DATA_BLOCK "G006G"
TITLE =
AUTHOR : KR
FAMILY : USW
VERSION : 0.0

"G006G_Code"
BEGIN
   Gr.FcCode := 0;
   Gr.Spare2 := 0;
   Gr.Spare4 := 0;
   Gr.Spare6 := 0;
   Gr.OutEmptyingTime := 0;
   Gr.ChangeBit.spare := B#16#0;
   Gr.ChangeBit.CBit1 := FALSE;
   Gr.ChangeBit.CBit2 := FALSE;
   Gr.ChangeBit.CBit3 := FALSE;
   Gr.ChangeBit.CBit4 := FALSE;
   Gr.StCode := 0;
   Gr.InEnableGr := FALSE;
   Gr.CmdContinue := FALSE;
   Gr.CmdRestartIdling := FALSE;
   Gr.InReleaseEmptyingTime := FALSE;
   Gr.InFeeding := FALSE;
   Gr.InOutAutostartMan := FALSE;
   Gr.InPreStart := FALSE;
   Gr.CmdManualOff := FALSE;
   Gr.CmdOff := FALSE;
   Gr.CmdOn := FALSE;
   Gr.CmdNext := FALSE;
   Gr.CmdFaultReset := FALSE;
   Gr.InOccupied := FALSE;
   Gr.InManual := FALSE;
   Gr.InLoadedSec := FALSE;
   Gr.InSeqStop := FALSE;
   Gr.ModePassive := FALSE;
   Gr.ModeActive := FALSE;
   Gr.ModeIdling := FALSE;
   Gr.spare163 := FALSE;
   Gr.spare164 := FALSE;
   Gr.spare165 := FALSE;
   Gr.spare166 := FALSE;
   Gr.spare167 := FALSE;
   Gr.StStopped := FALSE;
   Gr.StStarting := FALSE;
   Gr.StStarted := FALSE;
   Gr.StStopping := FALSE;
   Gr.StFault := FALSE;
   Gr.OutLoaded := FALSE;
   Gr.OutWarning := FALSE;
   Gr.OutFeeding := FALSE;
   Gr.OutEnableEl := FALSE;
   Gr.OutEnable1 := FALSE;
   Gr.OutHWStop := FALSE;
   Gr.OutDPFault := FALSE;
   Gr.OutAutostart := FALSE;
   Gr.OutManual := FALSE;
   Gr.OutHornOn := FALSE;
   Gr.OutEnablePrevGr := FALSE;
   Gr.VarStopped := FALSE;
   Gr.VarStarted := FALSE;
   Gr.VarFault := FALSE;
   Gr.VarStartwarning := FALSE;
   Gr.VarFlag1s := FALSE;
   Gr.OutEmptyingTimeDone := FALSE;
   Gr.OutNewWay := FALSE;
   Gr.OutSeqStop := FALSE;
   Gr.OutIdlingTime := 0;
   Gr.InCodePreselect := 0;
   Gr.InLine := 0;
   Gr.InCode := 0;
   Gr.OutCode := 0;
   Gr.Par.ParObjectNo := 0;
   Gr.Par.ParMgr := FALSE;
   Gr.Par.ParWgr := FALSE;
   Gr.Par.ParGgr := FALSE;
   Gr.Par.ParHornCode := 0;
   Gr.Par.ParIdling := 0;
   Gr.Par.ParEmptyingTime := 0;
   Gr.Par.Para1_0 := FALSE;
   Gr.Par.Para1_1 := FALSE;
   Gr.Par.Para1_2 := FALSE;
   Gr.Par.Para1_3 := FALSE;
   Gr.Par.Para1_4 := FALSE;
   Gr.Par.Para1_5 := FALSE;
   Gr.Par.Para1_6 := FALSE;
   Gr.Par.Para1_7 := FALSE;
   Gr.Par.Para1_8 := FALSE;
   Gr.Par.Para1_9 := FALSE;
   Gr.Par.Para1_10 := FALSE;
   Gr.Par.Para1_11 := FALSE;
   Gr.Par.Para1_12 := FALSE;
   Gr.Par.Para1_13 := FALSE;
   Gr.Par.Para1_14 := FALSE;
   Gr.Par.Para1_15 := FALSE;
   Gr.Par.Para2 := 0;
   Gr.Par.Para3 := 0;
   Gr.Par.Para4 := 0;
   Gr.Par.Para5 := 0;
   InOutValue1 := L#0;
   InOutValue2 := L#0;
   OutWayConflict := FALSE;
   OutSelectionOk := FALSE;
   CmdNewValue := FALSE;
   CmdNewJob := FALSE;
   OutCodeOK := FALSE;
   InEndOfJob := FALSE;
   staWayOk := FALSE;
   EdgeStartRelease := FALSE;
   USW8 := FALSE;
   USW9 := FALSE;
   USW10 := FALSE;
   USW11 := FALSE;
   USW12 := FALSE;
   USW13 := FALSE;
   USW14 := FALSE;
   USW15 := FALSE;
   A_1999_SHE01.StCode := 0;
   A_1999_SHE01.InMonTrue := FALSE;
   A_1999_SHE01.InMonFalse := FALSE;
   A_1999_SHE01.InPreAlarmTrue := FALSE;
   A_1999_SHE01.InPreAlarmFalse := FALSE;
   A_1999_SHE01.InStopTrueTime := FALSE;
   A_1999_SHE01.InStopFalseTime := FALSE;
   A_1999_SHE01.InpTrue := FALSE;
   A_1999_SHE01.InpFaultDev := FALSE;
   A_1999_SHE01.CmdRstTrueTime := FALSE;
   A_1999_SHE01.CmdRstFalseTime := FALSE;
   A_1999_SHE01.CmdRunTimeoutTime := FALSE;
   A_1999_SHE01.CmdFaultReset := FALSE;
   A_1999_SHE01.InLocal := FALSE;
   A_1999_SHE01.spare0305 := FALSE;
   A_1999_SHE01.InReport := FALSE;
   A_1999_SHE01.OutTimeoutTime := FALSE;
   A_1999_SHE01.InHWStop := FALSE;
   A_1999_SHE01.InDPFault := FALSE;
   A_1999_SHE01.OutPreAlarmTrue := FALSE;
   A_1999_SHE01.OutPreAlarmFalse := FALSE;
   A_1999_SHE01.OutFlagPos := FALSE;
   A_1999_SHE01.OutFlagNeg := FALSE;
   A_1999_SHE01.OutpFaultReset := FALSE;
   A_1999_SHE01.OutTrue := FALSE;
   A_1999_SHE01.StFalse := FALSE;
   A_1999_SHE01.StCtoTrue := FALSE;
   A_1999_SHE01.StTrue := FALSE;
   A_1999_SHE01.StCtoFalse := FALSE;
   A_1999_SHE01.StFault := FALSE;
   A_1999_SHE01.OutAlarmNrLog := 0;
   A_1999_SHE01.Par.ParObjectNo := 0;
   A_1999_SHE01.Par.ParMsgType := 0;
   A_1999_SHE01.Par.ParHornCode := 0;
   A_1999_SHE01.Par.ParLogOff := FALSE;
   A_1999_SHE01.Par.spare0401 := FALSE;
   A_1999_SHE01.Par.Par2WorkingCond := FALSE;
   A_1999_SHE01.Par.ParFaultRetry := FALSE;
   A_1999_SHE01.Par.ParBinLevel := FALSE;
   A_1999_SHE01.Par.ParDelayChange := 0;
   A_1999_SHE01.Par.ParDelayTrue := 0;
   A_1999_SHE01.Par.ParDelayFalse := 0;
   A_1999_SHE01.Par.ParTimeoutTrue := 0;
   A_1999_SHE01.Par.ParTimeoutFalse := 0;
   A_1999_SHE01.Par.OutMonTime := 0;
   A_1999_SHE01.Par.OutTransitionTime := 0;
   A_1999_SHE01.Par.OutMonTrue := FALSE;
   A_1999_SHE01.Par.OutMonFalse := FALSE;
   A_1999_SHE01.Par.OutFlagFaultDev := FALSE;
   A_1999_SHE01.Par.OutDelayTime := 0;
   A_1999_SHE02.StCode := 0;
   A_1999_SHE02.InMonTrue := FALSE;
   A_1999_SHE02.InMonFalse := FALSE;
   A_1999_SHE02.InPreAlarmTrue := FALSE;
   A_1999_SHE02.InPreAlarmFalse := FALSE;
   A_1999_SHE02.InStopTrueTime := FALSE;
   A_1999_SHE02.InStopFalseTime := FALSE;
   A_1999_SHE02.InpTrue := FALSE;
   A_1999_SHE02.InpFaultDev := FALSE;
   A_1999_SHE02.CmdRstTrueTime := FALSE;
   A_1999_SHE02.CmdRstFalseTime := FALSE;
   A_1999_SHE02.CmdRunTimeoutTime := FALSE;
   A_1999_SHE02.CmdFaultReset := FALSE;
   A_1999_SHE02.InLocal := FALSE;
   A_1999_SHE02.spare0305 := FALSE;
   A_1999_SHE02.InReport := FALSE;
   A_1999_SHE02.OutTimeoutTime := FALSE;
   A_1999_SHE02.InHWStop := FALSE;
   A_1999_SHE02.InDPFault := FALSE;
   A_1999_SHE02.OutPreAlarmTrue := FALSE;
   A_1999_SHE02.OutPreAlarmFalse := FALSE;
   A_1999_SHE02.OutFlagPos := FALSE;
   A_1999_SHE02.OutFlagNeg := FALSE;
   A_1999_SHE02.OutpFaultReset := FALSE;
   A_1999_SHE02.OutTrue := FALSE;
   A_1999_SHE02.StFalse := FALSE;
   A_1999_SHE02.StCtoTrue := FALSE;
   A_1999_SHE02.StTrue := FALSE;
   A_1999_SHE02.StCtoFalse := FALSE;
   A_1999_SHE02.StFault := FALSE;
   A_1999_SHE02.OutAlarmNrLog := 0;
   A_1999_SHE02.Par.ParObjectNo := 0;
   A_1999_SHE02.Par.ParMsgType := 0;
   A_1999_SHE02.Par.ParHornCode := 0;
   A_1999_SHE02.Par.ParLogOff := FALSE;
   A_1999_SHE02.Par.spare0401 := FALSE;
   A_1999_SHE02.Par.Par2WorkingCond := FALSE;
   A_1999_SHE02.Par.ParFaultRetry := FALSE;
   A_1999_SHE02.Par.ParBinLevel := FALSE;
   A_1999_SHE02.Par.ParDelayChange := 0;
   A_1999_SHE02.Par.ParDelayTrue := 0;
   A_1999_SHE02.Par.ParDelayFalse := 0;
   A_1999_SHE02.Par.ParTimeoutTrue := 0;
   A_1999_SHE02.Par.ParTimeoutFalse := 0;
   A_1999_SHE02.Par.OutMonTime := 0;
   A_1999_SHE02.Par.OutTransitionTime := 0;
   A_1999_SHE02.Par.OutMonTrue := FALSE;
   A_1999_SHE02.Par.OutMonFalse := FALSE;
   A_1999_SHE02.Par.OutFlagFaultDev := FALSE;
   A_1999_SHE02.Par.OutDelayTime := 0;
   A_19_A040Z1.StCode := 0;
   A_19_A040Z1.InMonTrue := FALSE;
   A_19_A040Z1.InMonFalse := FALSE;
   A_19_A040Z1.InPreAlarmTrue := FALSE;
   A_19_A040Z1.InPreAlarmFalse := FALSE;
   A_19_A040Z1.InStopTrueTime := FALSE;
   A_19_A040Z1.InStopFalseTime := FALSE;
   A_19_A040Z1.InpTrue := FALSE;
   A_19_A040Z1.InpFaultDev := FALSE;
   A_19_A040Z1.CmdRstTrueTime := FALSE;
   A_19_A040Z1.CmdRstFalseTime := FALSE;
   A_19_A040Z1.CmdRunTimeoutTime := FALSE;
   A_19_A040Z1.CmdFaultReset := FALSE;
   A_19_A040Z1.InLocal := FALSE;
   A_19_A040Z1.spare0305 := FALSE;
   A_19_A040Z1.InReport := FALSE;
   A_19_A040Z1.OutTimeoutTime := FALSE;
   A_19_A040Z1.InHWStop := FALSE;
   A_19_A040Z1.InDPFault := FALSE;
   A_19_A040Z1.OutPreAlarmTrue := FALSE;
   A_19_A040Z1.OutPreAlarmFalse := FALSE;
   A_19_A040Z1.OutFlagPos := FALSE;
   A_19_A040Z1.OutFlagNeg := FALSE;
   A_19_A040Z1.OutpFaultReset := FALSE;
   A_19_A040Z1.OutTrue := FALSE;
   A_19_A040Z1.StFalse := FALSE;
   A_19_A040Z1.StCtoTrue := FALSE;
   A_19_A040Z1.StTrue := FALSE;
   A_19_A040Z1.StCtoFalse := FALSE;
   A_19_A040Z1.StFault := FALSE;
   A_19_A040Z1.OutAlarmNrLog := 0;
   A_19_A040Z1.Par.ParObjectNo := 0;
   A_19_A040Z1.Par.ParMsgType := 0;
   A_19_A040Z1.Par.ParHornCode := 0;
   A_19_A040Z1.Par.ParLogOff := FALSE;
   A_19_A040Z1.Par.spare0401 := FALSE;
   A_19_A040Z1.Par.Par2WorkingCond := FALSE;
   A_19_A040Z1.Par.ParFaultRetry := FALSE;
   A_19_A040Z1.Par.ParBinLevel := FALSE;
   A_19_A040Z1.Par.ParDelayChange := 0;
   A_19_A040Z1.Par.ParDelayTrue := 0;
   A_19_A040Z1.Par.ParDelayFalse := 0;
   A_19_A040Z1.Par.ParTimeoutTrue := 0;
   A_19_A040Z1.Par.ParTimeoutFalse := 0;
   A_19_A040Z1.Par.OutMonTime := 0;
   A_19_A040Z1.Par.OutTransitionTime := 0;
   A_19_A040Z1.Par.OutMonTrue := FALSE;
   A_19_A040Z1.Par.OutMonFalse := FALSE;
   A_19_A040Z1.Par.OutFlagFaultDev := FALSE;
   A_19_A040Z1.Par.OutDelayTime := 0;
   A_19_A097Z1.StCode := 0;
   A_19_A097Z1.InMonTrue := FALSE;
   A_19_A097Z1.InMonFalse := FALSE;
   A_19_A097Z1.InPreAlarmTrue := FALSE;
   A_19_A097Z1.InPreAlarmFalse := FALSE;
   A_19_A097Z1.InStopTrueTime := FALSE;
   A_19_A097Z1.InStopFalseTime := FALSE;
   A_19_A097Z1.InpTrue := FALSE;
   A_19_A097Z1.InpFaultDev := FALSE;
   A_19_A097Z1.CmdRstTrueTime := FALSE;
   A_19_A097Z1.CmdRstFalseTime := FALSE;
   A_19_A097Z1.CmdRunTimeoutTime := FALSE;
   A_19_A097Z1.CmdFaultReset := FALSE;
   A_19_A097Z1.InLocal := FALSE;
   A_19_A097Z1.spare0305 := FALSE;
   A_19_A097Z1.InReport := FALSE;
   A_19_A097Z1.OutTimeoutTime := FALSE;
   A_19_A097Z1.InHWStop := FALSE;
   A_19_A097Z1.InDPFault := FALSE;
   A_19_A097Z1.OutPreAlarmTrue := FALSE;
   A_19_A097Z1.OutPreAlarmFalse := FALSE;
   A_19_A097Z1.OutFlagPos := FALSE;
   A_19_A097Z1.OutFlagNeg := FALSE;
   A_19_A097Z1.OutpFaultReset := FALSE;
   A_19_A097Z1.OutTrue := FALSE;
   A_19_A097Z1.StFalse := FALSE;
   A_19_A097Z1.StCtoTrue := FALSE;
   A_19_A097Z1.StTrue := FALSE;
   A_19_A097Z1.StCtoFalse := FALSE;
   A_19_A097Z1.StFault := FALSE;
   A_19_A097Z1.OutAlarmNrLog := 0;
   A_19_A097Z1.Par.ParObjectNo := 0;
   A_19_A097Z1.Par.ParMsgType := 0;
   A_19_A097Z1.Par.ParHornCode := 0;
   A_19_A097Z1.Par.ParLogOff := FALSE;
   A_19_A097Z1.Par.spare0401 := FALSE;
   A_19_A097Z1.Par.Par2WorkingCond := FALSE;
   A_19_A097Z1.Par.ParFaultRetry := FALSE;
   A_19_A097Z1.Par.ParBinLevel := FALSE;
   A_19_A097Z1.Par.ParDelayChange := 0;
   A_19_A097Z1.Par.ParDelayTrue := 0;
   A_19_A097Z1.Par.ParDelayFalse := 0;
   A_19_A097Z1.Par.ParTimeoutTrue := 0;
   A_19_A097Z1.Par.ParTimeoutFalse := 0;
   A_19_A097Z1.Par.OutMonTime := 0;
   A_19_A097Z1.Par.OutTransitionTime := 0;
   A_19_A097Z1.Par.OutMonTrue := FALSE;
   A_19_A097Z1.Par.OutMonFalse := FALSE;
   A_19_A097Z1.Par.OutFlagFaultDev := FALSE;
   A_19_A097Z1.Par.OutDelayTime := 0;
   A_19_K091Z1.StCode := 0;
   A_19_K091Z1.InMonTrue := FALSE;
   A_19_K091Z1.InMonFalse := FALSE;
   A_19_K091Z1.InPreAlarmTrue := FALSE;
   A_19_K091Z1.InPreAlarmFalse := FALSE;
   A_19_K091Z1.InStopTrueTime := FALSE;
   A_19_K091Z1.InStopFalseTime := FALSE;
   A_19_K091Z1.InpTrue := FALSE;
   A_19_K091Z1.InpFaultDev := FALSE;
   A_19_K091Z1.CmdRstTrueTime := FALSE;
   A_19_K091Z1.CmdRstFalseTime := FALSE;
   A_19_K091Z1.CmdRunTimeoutTime := FALSE;
   A_19_K091Z1.CmdFaultReset := FALSE;
   A_19_K091Z1.InLocal := FALSE;
   A_19_K091Z1.spare0305 := FALSE;
   A_19_K091Z1.InReport := FALSE;
   A_19_K091Z1.OutTimeoutTime := FALSE;
   A_19_K091Z1.InHWStop := FALSE;
   A_19_K091Z1.InDPFault := FALSE;
   A_19_K091Z1.OutPreAlarmTrue := FALSE;
   A_19_K091Z1.OutPreAlarmFalse := FALSE;
   A_19_K091Z1.OutFlagPos := FALSE;
   A_19_K091Z1.OutFlagNeg := FALSE;
   A_19_K091Z1.OutpFaultReset := FALSE;
   A_19_K091Z1.OutTrue := FALSE;
   A_19_K091Z1.StFalse := FALSE;
   A_19_K091Z1.StCtoTrue := FALSE;
   A_19_K091Z1.StTrue := FALSE;
   A_19_K091Z1.StCtoFalse := FALSE;
   A_19_K091Z1.StFault := FALSE;
   A_19_K091Z1.OutAlarmNrLog := 0;
   A_19_K091Z1.Par.ParObjectNo := 0;
   A_19_K091Z1.Par.ParMsgType := 0;
   A_19_K091Z1.Par.ParHornCode := 0;
   A_19_K091Z1.Par.ParLogOff := FALSE;
   A_19_K091Z1.Par.spare0401 := FALSE;
   A_19_K091Z1.Par.Par2WorkingCond := FALSE;
   A_19_K091Z1.Par.ParFaultRetry := FALSE;
   A_19_K091Z1.Par.ParBinLevel := FALSE;
   A_19_K091Z1.Par.ParDelayChange := 0;
   A_19_K091Z1.Par.ParDelayTrue := 0;
   A_19_K091Z1.Par.ParDelayFalse := 0;
   A_19_K091Z1.Par.ParTimeoutTrue := 0;
   A_19_K091Z1.Par.ParTimeoutFalse := 0;
   A_19_K091Z1.Par.OutMonTime := 0;
   A_19_K091Z1.Par.OutTransitionTime := 0;
   A_19_K091Z1.Par.OutMonTrue := FALSE;
   A_19_K091Z1.Par.OutMonFalse := FALSE;
   A_19_K091Z1.Par.OutFlagFaultDev := FALSE;
   A_19_K091Z1.Par.OutDelayTime := 0;
   A_19_S_H097Z1.StCode := 0;
   A_19_S_H097Z1.InMonTrue := FALSE;
   A_19_S_H097Z1.InMonFalse := FALSE;
   A_19_S_H097Z1.InPreAlarmTrue := FALSE;
   A_19_S_H097Z1.InPreAlarmFalse := FALSE;
   A_19_S_H097Z1.InStopTrueTime := FALSE;
   A_19_S_H097Z1.InStopFalseTime := FALSE;
   A_19_S_H097Z1.InpTrue := FALSE;
   A_19_S_H097Z1.InpFaultDev := FALSE;
   A_19_S_H097Z1.CmdRstTrueTime := FALSE;
   A_19_S_H097Z1.CmdRstFalseTime := FALSE;
   A_19_S_H097Z1.CmdRunTimeoutTime := FALSE;
   A_19_S_H097Z1.CmdFaultReset := FALSE;
   A_19_S_H097Z1.InLocal := FALSE;
   A_19_S_H097Z1.spare0305 := FALSE;
   A_19_S_H097Z1.InReport := FALSE;
   A_19_S_H097Z1.OutTimeoutTime := FALSE;
   A_19_S_H097Z1.InHWStop := FALSE;
   A_19_S_H097Z1.InDPFault := FALSE;
   A_19_S_H097Z1.OutPreAlarmTrue := FALSE;
   A_19_S_H097Z1.OutPreAlarmFalse := FALSE;
   A_19_S_H097Z1.OutFlagPos := FALSE;
   A_19_S_H097Z1.OutFlagNeg := FALSE;
   A_19_S_H097Z1.OutpFaultReset := FALSE;
   A_19_S_H097Z1.OutTrue := FALSE;
   A_19_S_H097Z1.StFalse := FALSE;
   A_19_S_H097Z1.StCtoTrue := FALSE;
   A_19_S_H097Z1.StTrue := FALSE;
   A_19_S_H097Z1.StCtoFalse := FALSE;
   A_19_S_H097Z1.StFault := FALSE;
   A_19_S_H097Z1.OutAlarmNrLog := 0;
   A_19_S_H097Z1.Par.ParObjectNo := 0;
   A_19_S_H097Z1.Par.ParMsgType := 0;
   A_19_S_H097Z1.Par.ParHornCode := 0;
   A_19_S_H097Z1.Par.ParLogOff := FALSE;
   A_19_S_H097Z1.Par.spare0401 := FALSE;
   A_19_S_H097Z1.Par.Par2WorkingCond := FALSE;
   A_19_S_H097Z1.Par.ParFaultRetry := FALSE;
   A_19_S_H097Z1.Par.ParBinLevel := FALSE;
   A_19_S_H097Z1.Par.ParDelayChange := 0;
   A_19_S_H097Z1.Par.ParDelayTrue := 0;
   A_19_S_H097Z1.Par.ParDelayFalse := 0;
   A_19_S_H097Z1.Par.ParTimeoutTrue := 0;
   A_19_S_H097Z1.Par.ParTimeoutFalse := 0;
   A_19_S_H097Z1.Par.OutMonTime := 0;
   A_19_S_H097Z1.Par.OutTransitionTime := 0;
   A_19_S_H097Z1.Par.OutMonTrue := FALSE;
   A_19_S_H097Z1.Par.OutMonFalse := FALSE;
   A_19_S_H097Z1.Par.OutFlagFaultDev := FALSE;
   A_19_S_H097Z1.Par.OutDelayTime := 0;
   A_2201_SHE20.StCode := 0;
   A_2201_SHE20.InMonTrue := FALSE;
   A_2201_SHE20.InMonFalse := FALSE;
   A_2201_SHE20.InPreAlarmTrue := FALSE;
   A_2201_SHE20.InPreAlarmFalse := FALSE;
   A_2201_SHE20.InStopTrueTime := FALSE;
   A_2201_SHE20.InStopFalseTime := FALSE;
   A_2201_SHE20.InpTrue := FALSE;
   A_2201_SHE20.InpFaultDev := FALSE;
   A_2201_SHE20.CmdRstTrueTime := FALSE;
   A_2201_SHE20.CmdRstFalseTime := FALSE;
   A_2201_SHE20.CmdRunTimeoutTime := FALSE;
   A_2201_SHE20.CmdFaultReset := FALSE;
   A_2201_SHE20.InLocal := FALSE;
   A_2201_SHE20.spare0305 := FALSE;
   A_2201_SHE20.InReport := FALSE;
   A_2201_SHE20.OutTimeoutTime := FALSE;
   A_2201_SHE20.InHWStop := FALSE;
   A_2201_SHE20.InDPFault := FALSE;
   A_2201_SHE20.OutPreAlarmTrue := FALSE;
   A_2201_SHE20.OutPreAlarmFalse := FALSE;
   A_2201_SHE20.OutFlagPos := FALSE;
   A_2201_SHE20.OutFlagNeg := FALSE;
   A_2201_SHE20.OutpFaultReset := FALSE;
   A_2201_SHE20.OutTrue := FALSE;
   A_2201_SHE20.StFalse := FALSE;
   A_2201_SHE20.StCtoTrue := FALSE;
   A_2201_SHE20.StTrue := FALSE;
   A_2201_SHE20.StCtoFalse := FALSE;
   A_2201_SHE20.StFault := FALSE;
   A_2201_SHE20.OutAlarmNrLog := 0;
   A_2201_SHE20.Par.ParObjectNo := 0;
   A_2201_SHE20.Par.ParMsgType := 0;
   A_2201_SHE20.Par.ParHornCode := 0;
   A_2201_SHE20.Par.ParLogOff := FALSE;
   A_2201_SHE20.Par.spare0401 := FALSE;
   A_2201_SHE20.Par.Par2WorkingCond := FALSE;
   A_2201_SHE20.Par.ParFaultRetry := FALSE;
   A_2201_SHE20.Par.ParBinLevel := FALSE;
   A_2201_SHE20.Par.ParDelayChange := 0;
   A_2201_SHE20.Par.ParDelayTrue := 0;
   A_2201_SHE20.Par.ParDelayFalse := 0;
   A_2201_SHE20.Par.ParTimeoutTrue := 0;
   A_2201_SHE20.Par.ParTimeoutFalse := 0;
   A_2201_SHE20.Par.OutMonTime := 0;
   A_2201_SHE20.Par.OutTransitionTime := 0;
   A_2201_SHE20.Par.OutMonTrue := FALSE;
   A_2201_SHE20.Par.OutMonFalse := FALSE;
   A_2201_SHE20.Par.OutFlagFaultDev := FALSE;
   A_2201_SHE20.Par.OutDelayTime := 0;
   A_2201_SHE21.StCode := 0;
   A_2201_SHE21.InMonTrue := FALSE;
   A_2201_SHE21.InMonFalse := FALSE;
   A_2201_SHE21.InPreAlarmTrue := FALSE;
   A_2201_SHE21.InPreAlarmFalse := FALSE;
   A_2201_SHE21.InStopTrueTime := FALSE;
   A_2201_SHE21.InStopFalseTime := FALSE;
   A_2201_SHE21.InpTrue := FALSE;
   A_2201_SHE21.InpFaultDev := FALSE;
   A_2201_SHE21.CmdRstTrueTime := FALSE;
   A_2201_SHE21.CmdRstFalseTime := FALSE;
   A_2201_SHE21.CmdRunTimeoutTime := FALSE;
   A_2201_SHE21.CmdFaultReset := FALSE;
   A_2201_SHE21.InLocal := FALSE;
   A_2201_SHE21.spare0305 := FALSE;
   A_2201_SHE21.InReport := FALSE;
   A_2201_SHE21.OutTimeoutTime := FALSE;
   A_2201_SHE21.InHWStop := FALSE;
   A_2201_SHE21.InDPFault := FALSE;
   A_2201_SHE21.OutPreAlarmTrue := FALSE;
   A_2201_SHE21.OutPreAlarmFalse := FALSE;
   A_2201_SHE21.OutFlagPos := FALSE;
   A_2201_SHE21.OutFlagNeg := FALSE;
   A_2201_SHE21.OutpFaultReset := FALSE;
   A_2201_SHE21.OutTrue := FALSE;
   A_2201_SHE21.StFalse := FALSE;
   A_2201_SHE21.StCtoTrue := FALSE;
   A_2201_SHE21.StTrue := FALSE;
   A_2201_SHE21.StCtoFalse := FALSE;
   A_2201_SHE21.StFault := FALSE;
   A_2201_SHE21.OutAlarmNrLog := 0;
   A_2201_SHE21.Par.ParObjectNo := 0;
   A_2201_SHE21.Par.ParMsgType := 0;
   A_2201_SHE21.Par.ParHornCode := 0;
   A_2201_SHE21.Par.ParLogOff := FALSE;
   A_2201_SHE21.Par.spare0401 := FALSE;
   A_2201_SHE21.Par.Par2WorkingCond := FALSE;
   A_2201_SHE21.Par.ParFaultRetry := FALSE;
   A_2201_SHE21.Par.ParBinLevel := FALSE;
   A_2201_SHE21.Par.ParDelayChange := 0;
   A_2201_SHE21.Par.ParDelayTrue := 0;
   A_2201_SHE21.Par.ParDelayFalse := 0;
   A_2201_SHE21.Par.ParTimeoutTrue := 0;
   A_2201_SHE21.Par.ParTimeoutFalse := 0;
   A_2201_SHE21.Par.OutMonTime := 0;
   A_2201_SHE21.Par.OutTransitionTime := 0;
   A_2201_SHE21.Par.OutMonTrue := FALSE;
   A_2201_SHE21.Par.OutMonFalse := FALSE;
   A_2201_SHE21.Par.OutFlagFaultDev := FALSE;
   A_2201_SHE21.Par.OutDelayTime := 0;
   A_2201_SHE22.StCode := 0;
   A_2201_SHE22.InMonTrue := FALSE;
   A_2201_SHE22.InMonFalse := FALSE;
   A_2201_SHE22.InPreAlarmTrue := FALSE;
   A_2201_SHE22.InPreAlarmFalse := FALSE;
   A_2201_SHE22.InStopTrueTime := FALSE;
   A_2201_SHE22.InStopFalseTime := FALSE;
   A_2201_SHE22.InpTrue := FALSE;
   A_2201_SHE22.InpFaultDev := FALSE;
   A_2201_SHE22.CmdRstTrueTime := FALSE;
   A_2201_SHE22.CmdRstFalseTime := FALSE;
   A_2201_SHE22.CmdRunTimeoutTime := FALSE;
   A_2201_SHE22.CmdFaultReset := FALSE;
   A_2201_SHE22.InLocal := FALSE;
   A_2201_SHE22.spare0305 := FALSE;
   A_2201_SHE22.InReport := FALSE;
   A_2201_SHE22.OutTimeoutTime := FALSE;
   A_2201_SHE22.InHWStop := FALSE;
   A_2201_SHE22.InDPFault := FALSE;
   A_2201_SHE22.OutPreAlarmTrue := FALSE;
   A_2201_SHE22.OutPreAlarmFalse := FALSE;
   A_2201_SHE22.OutFlagPos := FALSE;
   A_2201_SHE22.OutFlagNeg := FALSE;
   A_2201_SHE22.OutpFaultReset := FALSE;
   A_2201_SHE22.OutTrue := FALSE;
   A_2201_SHE22.StFalse := FALSE;
   A_2201_SHE22.StCtoTrue := FALSE;
   A_2201_SHE22.StTrue := FALSE;
   A_2201_SHE22.StCtoFalse := FALSE;
   A_2201_SHE22.StFault := FALSE;
   A_2201_SHE22.OutAlarmNrLog := 0;
   A_2201_SHE22.Par.ParObjectNo := 0;
   A_2201_SHE22.Par.ParMsgType := 0;
   A_2201_SHE22.Par.ParHornCode := 0;
   A_2201_SHE22.Par.ParLogOff := FALSE;
   A_2201_SHE22.Par.spare0401 := FALSE;
   A_2201_SHE22.Par.Par2WorkingCond := FALSE;
   A_2201_SHE22.Par.ParFaultRetry := FALSE;
   A_2201_SHE22.Par.ParBinLevel := FALSE;
   A_2201_SHE22.Par.ParDelayChange := 0;
   A_2201_SHE22.Par.ParDelayTrue := 0;
   A_2201_SHE22.Par.ParDelayFalse := 0;
   A_2201_SHE22.Par.ParTimeoutTrue := 0;
   A_2201_SHE22.Par.ParTimeoutFalse := 0;
   A_2201_SHE22.Par.OutMonTime := 0;
   A_2201_SHE22.Par.OutTransitionTime := 0;
   A_2201_SHE22.Par.OutMonTrue := FALSE;
   A_2201_SHE22.Par.OutMonFalse := FALSE;
   A_2201_SHE22.Par.OutFlagFaultDev := FALSE;
   A_2201_SHE22.Par.OutDelayTime := 0;
   A_2201_SHE23.StCode := 0;
   A_2201_SHE23.InMonTrue := FALSE;
   A_2201_SHE23.InMonFalse := FALSE;
   A_2201_SHE23.InPreAlarmTrue := FALSE;
   A_2201_SHE23.InPreAlarmFalse := FALSE;
   A_2201_SHE23.InStopTrueTime := FALSE;
   A_2201_SHE23.InStopFalseTime := FALSE;
   A_2201_SHE23.InpTrue := FALSE;
   A_2201_SHE23.InpFaultDev := FALSE;
   A_2201_SHE23.CmdRstTrueTime := FALSE;
   A_2201_SHE23.CmdRstFalseTime := FALSE;
   A_2201_SHE23.CmdRunTimeoutTime := FALSE;
   A_2201_SHE23.CmdFaultReset := FALSE;
   A_2201_SHE23.InLocal := FALSE;
   A_2201_SHE23.spare0305 := FALSE;
   A_2201_SHE23.InReport := FALSE;
   A_2201_SHE23.OutTimeoutTime := FALSE;
   A_2201_SHE23.InHWStop := FALSE;
   A_2201_SHE23.InDPFault := FALSE;
   A_2201_SHE23.OutPreAlarmTrue := FALSE;
   A_2201_SHE23.OutPreAlarmFalse := FALSE;
   A_2201_SHE23.OutFlagPos := FALSE;
   A_2201_SHE23.OutFlagNeg := FALSE;
   A_2201_SHE23.OutpFaultReset := FALSE;
   A_2201_SHE23.OutTrue := FALSE;
   A_2201_SHE23.StFalse := FALSE;
   A_2201_SHE23.StCtoTrue := FALSE;
   A_2201_SHE23.StTrue := FALSE;
   A_2201_SHE23.StCtoFalse := FALSE;
   A_2201_SHE23.StFault := FALSE;
   A_2201_SHE23.OutAlarmNrLog := 0;
   A_2201_SHE23.Par.ParObjectNo := 0;
   A_2201_SHE23.Par.ParMsgType := 0;
   A_2201_SHE23.Par.ParHornCode := 0;
   A_2201_SHE23.Par.ParLogOff := FALSE;
   A_2201_SHE23.Par.spare0401 := FALSE;
   A_2201_SHE23.Par.Par2WorkingCond := FALSE;
   A_2201_SHE23.Par.ParFaultRetry := FALSE;
   A_2201_SHE23.Par.ParBinLevel := FALSE;
   A_2201_SHE23.Par.ParDelayChange := 0;
   A_2201_SHE23.Par.ParDelayTrue := 0;
   A_2201_SHE23.Par.ParDelayFalse := 0;
   A_2201_SHE23.Par.ParTimeoutTrue := 0;
   A_2201_SHE23.Par.ParTimeoutFalse := 0;
   A_2201_SHE23.Par.OutMonTime := 0;
   A_2201_SHE23.Par.OutTransitionTime := 0;
   A_2201_SHE23.Par.OutMonTrue := FALSE;
   A_2201_SHE23.Par.OutMonFalse := FALSE;
   A_2201_SHE23.Par.OutFlagFaultDev := FALSE;
   A_2201_SHE23.Par.OutDelayTime := 0;
   A_2299_SHE01.StCode := 0;
   A_2299_SHE01.InMonTrue := FALSE;
   A_2299_SHE01.InMonFalse := FALSE;
   A_2299_SHE01.InPreAlarmTrue := FALSE;
   A_2299_SHE01.InPreAlarmFalse := FALSE;
   A_2299_SHE01.InStopTrueTime := FALSE;
   A_2299_SHE01.InStopFalseTime := FALSE;
   A_2299_SHE01.InpTrue := FALSE;
   A_2299_SHE01.InpFaultDev := FALSE;
   A_2299_SHE01.CmdRstTrueTime := FALSE;
   A_2299_SHE01.CmdRstFalseTime := FALSE;
   A_2299_SHE01.CmdRunTimeoutTime := FALSE;
   A_2299_SHE01.CmdFaultReset := FALSE;
   A_2299_SHE01.InLocal := FALSE;
   A_2299_SHE01.spare0305 := FALSE;
   A_2299_SHE01.InReport := FALSE;
   A_2299_SHE01.OutTimeoutTime := FALSE;
   A_2299_SHE01.InHWStop := FALSE;
   A_2299_SHE01.InDPFault := FALSE;
   A_2299_SHE01.OutPreAlarmTrue := FALSE;
   A_2299_SHE01.OutPreAlarmFalse := FALSE;
   A_2299_SHE01.OutFlagPos := FALSE;
   A_2299_SHE01.OutFlagNeg := FALSE;
   A_2299_SHE01.OutpFaultReset := FALSE;
   A_2299_SHE01.OutTrue := FALSE;
   A_2299_SHE01.StFalse := FALSE;
   A_2299_SHE01.StCtoTrue := FALSE;
   A_2299_SHE01.StTrue := FALSE;
   A_2299_SHE01.StCtoFalse := FALSE;
   A_2299_SHE01.StFault := FALSE;
   A_2299_SHE01.OutAlarmNrLog := 0;
   A_2299_SHE01.Par.ParObjectNo := 0;
   A_2299_SHE01.Par.ParMsgType := 0;
   A_2299_SHE01.Par.ParHornCode := 0;
   A_2299_SHE01.Par.ParLogOff := FALSE;
   A_2299_SHE01.Par.spare0401 := FALSE;
   A_2299_SHE01.Par.Par2WorkingCond := FALSE;
   A_2299_SHE01.Par.ParFaultRetry := FALSE;
   A_2299_SHE01.Par.ParBinLevel := FALSE;
   A_2299_SHE01.Par.ParDelayChange := 0;
   A_2299_SHE01.Par.ParDelayTrue := 0;
   A_2299_SHE01.Par.ParDelayFalse := 0;
   A_2299_SHE01.Par.ParTimeoutTrue := 0;
   A_2299_SHE01.Par.ParTimeoutFalse := 0;
   A_2299_SHE01.Par.OutMonTime := 0;
   A_2299_SHE01.Par.OutTransitionTime := 0;
   A_2299_SHE01.Par.OutMonTrue := FALSE;
   A_2299_SHE01.Par.OutMonFalse := FALSE;
   A_2299_SHE01.Par.OutFlagFaultDev := FALSE;
   A_2299_SHE01.Par.OutDelayTime := 0;
   A_2299_SHE02.StCode := 0;
   A_2299_SHE02.InMonTrue := FALSE;
   A_2299_SHE02.InMonFalse := FALSE;
   A_2299_SHE02.InPreAlarmTrue := FALSE;
   A_2299_SHE02.InPreAlarmFalse := FALSE;
   A_2299_SHE02.InStopTrueTime := FALSE;
   A_2299_SHE02.InStopFalseTime := FALSE;
   A_2299_SHE02.InpTrue := FALSE;
   A_2299_SHE02.InpFaultDev := FALSE;
   A_2299_SHE02.CmdRstTrueTime := FALSE;
   A_2299_SHE02.CmdRstFalseTime := FALSE;
   A_2299_SHE02.CmdRunTimeoutTime := FALSE;
   A_2299_SHE02.CmdFaultReset := FALSE;
   A_2299_SHE02.InLocal := FALSE;
   A_2299_SHE02.spare0305 := FALSE;
   A_2299_SHE02.InReport := FALSE;
   A_2299_SHE02.OutTimeoutTime := FALSE;
   A_2299_SHE02.InHWStop := FALSE;
   A_2299_SHE02.InDPFault := FALSE;
   A_2299_SHE02.OutPreAlarmTrue := FALSE;
   A_2299_SHE02.OutPreAlarmFalse := FALSE;
   A_2299_SHE02.OutFlagPos := FALSE;
   A_2299_SHE02.OutFlagNeg := FALSE;
   A_2299_SHE02.OutpFaultReset := FALSE;
   A_2299_SHE02.OutTrue := FALSE;
   A_2299_SHE02.StFalse := FALSE;
   A_2299_SHE02.StCtoTrue := FALSE;
   A_2299_SHE02.StTrue := FALSE;
   A_2299_SHE02.StCtoFalse := FALSE;
   A_2299_SHE02.StFault := FALSE;
   A_2299_SHE02.OutAlarmNrLog := 0;
   A_2299_SHE02.Par.ParObjectNo := 0;
   A_2299_SHE02.Par.ParMsgType := 0;
   A_2299_SHE02.Par.ParHornCode := 0;
   A_2299_SHE02.Par.ParLogOff := FALSE;
   A_2299_SHE02.Par.spare0401 := FALSE;
   A_2299_SHE02.Par.Par2WorkingCond := FALSE;
   A_2299_SHE02.Par.ParFaultRetry := FALSE;
   A_2299_SHE02.Par.ParBinLevel := FALSE;
   A_2299_SHE02.Par.ParDelayChange := 0;
   A_2299_SHE02.Par.ParDelayTrue := 0;
   A_2299_SHE02.Par.ParDelayFalse := 0;
   A_2299_SHE02.Par.ParTimeoutTrue := 0;
   A_2299_SHE02.Par.ParTimeoutFalse := 0;
   A_2299_SHE02.Par.OutMonTime := 0;
   A_2299_SHE02.Par.OutTransitionTime := 0;
   A_2299_SHE02.Par.OutMonTrue := FALSE;
   A_2299_SHE02.Par.OutMonFalse := FALSE;
   A_2299_SHE02.Par.OutFlagFaultDev := FALSE;
   A_2299_SHE02.Par.OutDelayTime := 0;
   A_2299_SHE03.StCode := 0;
   A_2299_SHE03.InMonTrue := FALSE;
   A_2299_SHE03.InMonFalse := FALSE;
   A_2299_SHE03.InPreAlarmTrue := FALSE;
   A_2299_SHE03.InPreAlarmFalse := FALSE;
   A_2299_SHE03.InStopTrueTime := FALSE;
   A_2299_SHE03.InStopFalseTime := FALSE;
   A_2299_SHE03.InpTrue := FALSE;
   A_2299_SHE03.InpFaultDev := FALSE;
   A_2299_SHE03.CmdRstTrueTime := FALSE;
   A_2299_SHE03.CmdRstFalseTime := FALSE;
   A_2299_SHE03.CmdRunTimeoutTime := FALSE;
   A_2299_SHE03.CmdFaultReset := FALSE;
   A_2299_SHE03.InLocal := FALSE;
   A_2299_SHE03.spare0305 := FALSE;
   A_2299_SHE03.InReport := FALSE;
   A_2299_SHE03.OutTimeoutTime := FALSE;
   A_2299_SHE03.InHWStop := FALSE;
   A_2299_SHE03.InDPFault := FALSE;
   A_2299_SHE03.OutPreAlarmTrue := FALSE;
   A_2299_SHE03.OutPreAlarmFalse := FALSE;
   A_2299_SHE03.OutFlagPos := FALSE;
   A_2299_SHE03.OutFlagNeg := FALSE;
   A_2299_SHE03.OutpFaultReset := FALSE;
   A_2299_SHE03.OutTrue := FALSE;
   A_2299_SHE03.StFalse := FALSE;
   A_2299_SHE03.StCtoTrue := FALSE;
   A_2299_SHE03.StTrue := FALSE;
   A_2299_SHE03.StCtoFalse := FALSE;
   A_2299_SHE03.StFault := FALSE;
   A_2299_SHE03.OutAlarmNrLog := 0;
   A_2299_SHE03.Par.ParObjectNo := 0;
   A_2299_SHE03.Par.ParMsgType := 0;
   A_2299_SHE03.Par.ParHornCode := 0;
   A_2299_SHE03.Par.ParLogOff := FALSE;
   A_2299_SHE03.Par.spare0401 := FALSE;
   A_2299_SHE03.Par.Par2WorkingCond := FALSE;
   A_2299_SHE03.Par.ParFaultRetry := FALSE;
   A_2299_SHE03.Par.ParBinLevel := FALSE;
   A_2299_SHE03.Par.ParDelayChange := 0;
   A_2299_SHE03.Par.ParDelayTrue := 0;
   A_2299_SHE03.Par.ParDelayFalse := 0;
   A_2299_SHE03.Par.ParTimeoutTrue := 0;
   A_2299_SHE03.Par.ParTimeoutFalse := 0;
   A_2299_SHE03.Par.OutMonTime := 0;
   A_2299_SHE03.Par.OutTransitionTime := 0;
   A_2299_SHE03.Par.OutMonTrue := FALSE;
   A_2299_SHE03.Par.OutMonFalse := FALSE;
   A_2299_SHE03.Par.OutFlagFaultDev := FALSE;
   A_2299_SHE03.Par.OutDelayTime := 0;
   A_2299_SHE04.StCode := 0;
   A_2299_SHE04.InMonTrue := FALSE;
   A_2299_SHE04.InMonFalse := FALSE;
   A_2299_SHE04.InPreAlarmTrue := FALSE;
   A_2299_SHE04.InPreAlarmFalse := FALSE;
   A_2299_SHE04.InStopTrueTime := FALSE;
   A_2299_SHE04.InStopFalseTime := FALSE;
   A_2299_SHE04.InpTrue := FALSE;
   A_2299_SHE04.InpFaultDev := FALSE;
   A_2299_SHE04.CmdRstTrueTime := FALSE;
   A_2299_SHE04.CmdRstFalseTime := FALSE;
   A_2299_SHE04.CmdRunTimeoutTime := FALSE;
   A_2299_SHE04.CmdFaultReset := FALSE;
   A_2299_SHE04.InLocal := FALSE;
   A_2299_SHE04.spare0305 := FALSE;
   A_2299_SHE04.InReport := FALSE;
   A_2299_SHE04.OutTimeoutTime := FALSE;
   A_2299_SHE04.InHWStop := FALSE;
   A_2299_SHE04.InDPFault := FALSE;
   A_2299_SHE04.OutPreAlarmTrue := FALSE;
   A_2299_SHE04.OutPreAlarmFalse := FALSE;
   A_2299_SHE04.OutFlagPos := FALSE;
   A_2299_SHE04.OutFlagNeg := FALSE;
   A_2299_SHE04.OutpFaultReset := FALSE;
   A_2299_SHE04.OutTrue := FALSE;
   A_2299_SHE04.StFalse := FALSE;
   A_2299_SHE04.StCtoTrue := FALSE;
   A_2299_SHE04.StTrue := FALSE;
   A_2299_SHE04.StCtoFalse := FALSE;
   A_2299_SHE04.StFault := FALSE;
   A_2299_SHE04.OutAlarmNrLog := 0;
   A_2299_SHE04.Par.ParObjectNo := 0;
   A_2299_SHE04.Par.ParMsgType := 0;
   A_2299_SHE04.Par.ParHornCode := 0;
   A_2299_SHE04.Par.ParLogOff := FALSE;
   A_2299_SHE04.Par.spare0401 := FALSE;
   A_2299_SHE04.Par.Par2WorkingCond := FALSE;
   A_2299_SHE04.Par.ParFaultRetry := FALSE;
   A_2299_SHE04.Par.ParBinLevel := FALSE;
   A_2299_SHE04.Par.ParDelayChange := 0;
   A_2299_SHE04.Par.ParDelayTrue := 0;
   A_2299_SHE04.Par.ParDelayFalse := 0;
   A_2299_SHE04.Par.ParTimeoutTrue := 0;
   A_2299_SHE04.Par.ParTimeoutFalse := 0;
   A_2299_SHE04.Par.OutMonTime := 0;
   A_2299_SHE04.Par.OutTransitionTime := 0;
   A_2299_SHE04.Par.OutMonTrue := FALSE;
   A_2299_SHE04.Par.OutMonFalse := FALSE;
   A_2299_SHE04.Par.OutFlagFaultDev := FALSE;
   A_2299_SHE04.Par.OutDelayTime := 0;
   A_2299_SHE05.StCode := 0;
   A_2299_SHE05.InMonTrue := FALSE;
   A_2299_SHE05.InMonFalse := FALSE;
   A_2299_SHE05.InPreAlarmTrue := FALSE;
   A_2299_SHE05.InPreAlarmFalse := FALSE;
   A_2299_SHE05.InStopTrueTime := FALSE;
   A_2299_SHE05.InStopFalseTime := FALSE;
   A_2299_SHE05.InpTrue := FALSE;
   A_2299_SHE05.InpFaultDev := FALSE;
   A_2299_SHE05.CmdRstTrueTime := FALSE;
   A_2299_SHE05.CmdRstFalseTime := FALSE;
   A_2299_SHE05.CmdRunTimeoutTime := FALSE;
   A_2299_SHE05.CmdFaultReset := FALSE;
   A_2299_SHE05.InLocal := FALSE;
   A_2299_SHE05.spare0305 := FALSE;
   A_2299_SHE05.InReport := FALSE;
   A_2299_SHE05.OutTimeoutTime := FALSE;
   A_2299_SHE05.InHWStop := FALSE;
   A_2299_SHE05.InDPFault := FALSE;
   A_2299_SHE05.OutPreAlarmTrue := FALSE;
   A_2299_SHE05.OutPreAlarmFalse := FALSE;
   A_2299_SHE05.OutFlagPos := FALSE;
   A_2299_SHE05.OutFlagNeg := FALSE;
   A_2299_SHE05.OutpFaultReset := FALSE;
   A_2299_SHE05.OutTrue := FALSE;
   A_2299_SHE05.StFalse := FALSE;
   A_2299_SHE05.StCtoTrue := FALSE;
   A_2299_SHE05.StTrue := FALSE;
   A_2299_SHE05.StCtoFalse := FALSE;
   A_2299_SHE05.StFault := FALSE;
   A_2299_SHE05.OutAlarmNrLog := 0;
   A_2299_SHE05.Par.ParObjectNo := 0;
   A_2299_SHE05.Par.ParMsgType := 0;
   A_2299_SHE05.Par.ParHornCode := 0;
   A_2299_SHE05.Par.ParLogOff := FALSE;
   A_2299_SHE05.Par.spare0401 := FALSE;
   A_2299_SHE05.Par.Par2WorkingCond := FALSE;
   A_2299_SHE05.Par.ParFaultRetry := FALSE;
   A_2299_SHE05.Par.ParBinLevel := FALSE;
   A_2299_SHE05.Par.ParDelayChange := 0;
   A_2299_SHE05.Par.ParDelayTrue := 0;
   A_2299_SHE05.Par.ParDelayFalse := 0;
   A_2299_SHE05.Par.ParTimeoutTrue := 0;
   A_2299_SHE05.Par.ParTimeoutFalse := 0;
   A_2299_SHE05.Par.OutMonTime := 0;
   A_2299_SHE05.Par.OutTransitionTime := 0;
   A_2299_SHE05.Par.OutMonTrue := FALSE;
   A_2299_SHE05.Par.OutMonFalse := FALSE;
   A_2299_SHE05.Par.OutFlagFaultDev := FALSE;
   A_2299_SHE05.Par.OutDelayTime := 0;
   A_2299_SHE06.StCode := 0;
   A_2299_SHE06.InMonTrue := FALSE;
   A_2299_SHE06.InMonFalse := FALSE;
   A_2299_SHE06.InPreAlarmTrue := FALSE;
   A_2299_SHE06.InPreAlarmFalse := FALSE;
   A_2299_SHE06.InStopTrueTime := FALSE;
   A_2299_SHE06.InStopFalseTime := FALSE;
   A_2299_SHE06.InpTrue := FALSE;
   A_2299_SHE06.InpFaultDev := FALSE;
   A_2299_SHE06.CmdRstTrueTime := FALSE;
   A_2299_SHE06.CmdRstFalseTime := FALSE;
   A_2299_SHE06.CmdRunTimeoutTime := FALSE;
   A_2299_SHE06.CmdFaultReset := FALSE;
   A_2299_SHE06.InLocal := FALSE;
   A_2299_SHE06.spare0305 := FALSE;
   A_2299_SHE06.InReport := FALSE;
   A_2299_SHE06.OutTimeoutTime := FALSE;
   A_2299_SHE06.InHWStop := FALSE;
   A_2299_SHE06.InDPFault := FALSE;
   A_2299_SHE06.OutPreAlarmTrue := FALSE;
   A_2299_SHE06.OutPreAlarmFalse := FALSE;
   A_2299_SHE06.OutFlagPos := FALSE;
   A_2299_SHE06.OutFlagNeg := FALSE;
   A_2299_SHE06.OutpFaultReset := FALSE;
   A_2299_SHE06.OutTrue := FALSE;
   A_2299_SHE06.StFalse := FALSE;
   A_2299_SHE06.StCtoTrue := FALSE;
   A_2299_SHE06.StTrue := FALSE;
   A_2299_SHE06.StCtoFalse := FALSE;
   A_2299_SHE06.StFault := FALSE;
   A_2299_SHE06.OutAlarmNrLog := 0;
   A_2299_SHE06.Par.ParObjectNo := 0;
   A_2299_SHE06.Par.ParMsgType := 0;
   A_2299_SHE06.Par.ParHornCode := 0;
   A_2299_SHE06.Par.ParLogOff := FALSE;
   A_2299_SHE06.Par.spare0401 := FALSE;
   A_2299_SHE06.Par.Par2WorkingCond := FALSE;
   A_2299_SHE06.Par.ParFaultRetry := FALSE;
   A_2299_SHE06.Par.ParBinLevel := FALSE;
   A_2299_SHE06.Par.ParDelayChange := 0;
   A_2299_SHE06.Par.ParDelayTrue := 0;
   A_2299_SHE06.Par.ParDelayFalse := 0;
   A_2299_SHE06.Par.ParTimeoutTrue := 0;
   A_2299_SHE06.Par.ParTimeoutFalse := 0;
   A_2299_SHE06.Par.OutMonTime := 0;
   A_2299_SHE06.Par.OutTransitionTime := 0;
   A_2299_SHE06.Par.OutMonTrue := FALSE;
   A_2299_SHE06.Par.OutMonFalse := FALSE;
   A_2299_SHE06.Par.OutFlagFaultDev := FALSE;
   A_2299_SHE06.Par.OutDelayTime := 0;
   A_2299_SHE08.StCode := 0;
   A_2299_SHE08.InMonTrue := FALSE;
   A_2299_SHE08.InMonFalse := FALSE;
   A_2299_SHE08.InPreAlarmTrue := FALSE;
   A_2299_SHE08.InPreAlarmFalse := FALSE;
   A_2299_SHE08.InStopTrueTime := FALSE;
   A_2299_SHE08.InStopFalseTime := FALSE;
   A_2299_SHE08.InpTrue := FALSE;
   A_2299_SHE08.InpFaultDev := FALSE;
   A_2299_SHE08.CmdRstTrueTime := FALSE;
   A_2299_SHE08.CmdRstFalseTime := FALSE;
   A_2299_SHE08.CmdRunTimeoutTime := FALSE;
   A_2299_SHE08.CmdFaultReset := FALSE;
   A_2299_SHE08.InLocal := FALSE;
   A_2299_SHE08.spare0305 := FALSE;
   A_2299_SHE08.InReport := FALSE;
   A_2299_SHE08.OutTimeoutTime := FALSE;
   A_2299_SHE08.InHWStop := FALSE;
   A_2299_SHE08.InDPFault := FALSE;
   A_2299_SHE08.OutPreAlarmTrue := FALSE;
   A_2299_SHE08.OutPreAlarmFalse := FALSE;
   A_2299_SHE08.OutFlagPos := FALSE;
   A_2299_SHE08.OutFlagNeg := FALSE;
   A_2299_SHE08.OutpFaultReset := FALSE;
   A_2299_SHE08.OutTrue := FALSE;
   A_2299_SHE08.StFalse := FALSE;
   A_2299_SHE08.StCtoTrue := FALSE;
   A_2299_SHE08.StTrue := FALSE;
   A_2299_SHE08.StCtoFalse := FALSE;
   A_2299_SHE08.StFault := FALSE;
   A_2299_SHE08.OutAlarmNrLog := 0;
   A_2299_SHE08.Par.ParObjectNo := 0;
   A_2299_SHE08.Par.ParMsgType := 0;
   A_2299_SHE08.Par.ParHornCode := 0;
   A_2299_SHE08.Par.ParLogOff := FALSE;
   A_2299_SHE08.Par.spare0401 := FALSE;
   A_2299_SHE08.Par.Par2WorkingCond := FALSE;
   A_2299_SHE08.Par.ParFaultRetry := FALSE;
   A_2299_SHE08.Par.ParBinLevel := FALSE;
   A_2299_SHE08.Par.ParDelayChange := 0;
   A_2299_SHE08.Par.ParDelayTrue := 0;
   A_2299_SHE08.Par.ParDelayFalse := 0;
   A_2299_SHE08.Par.ParTimeoutTrue := 0;
   A_2299_SHE08.Par.ParTimeoutFalse := 0;
   A_2299_SHE08.Par.OutMonTime := 0;
   A_2299_SHE08.Par.OutTransitionTime := 0;
   A_2299_SHE08.Par.OutMonTrue := FALSE;
   A_2299_SHE08.Par.OutMonFalse := FALSE;
   A_2299_SHE08.Par.OutFlagFaultDev := FALSE;
   A_2299_SHE08.Par.OutDelayTime := 0;
   A_2299_SHE20.StCode := 0;
   A_2299_SHE20.InMonTrue := FALSE;
   A_2299_SHE20.InMonFalse := FALSE;
   A_2299_SHE20.InPreAlarmTrue := FALSE;
   A_2299_SHE20.InPreAlarmFalse := FALSE;
   A_2299_SHE20.InStopTrueTime := FALSE;
   A_2299_SHE20.InStopFalseTime := FALSE;
   A_2299_SHE20.InpTrue := FALSE;
   A_2299_SHE20.InpFaultDev := FALSE;
   A_2299_SHE20.CmdRstTrueTime := FALSE;
   A_2299_SHE20.CmdRstFalseTime := FALSE;
   A_2299_SHE20.CmdRunTimeoutTime := FALSE;
   A_2299_SHE20.CmdFaultReset := FALSE;
   A_2299_SHE20.InLocal := FALSE;
   A_2299_SHE20.spare0305 := FALSE;
   A_2299_SHE20.InReport := FALSE;
   A_2299_SHE20.OutTimeoutTime := FALSE;
   A_2299_SHE20.InHWStop := FALSE;
   A_2299_SHE20.InDPFault := FALSE;
   A_2299_SHE20.OutPreAlarmTrue := FALSE;
   A_2299_SHE20.OutPreAlarmFalse := FALSE;
   A_2299_SHE20.OutFlagPos := FALSE;
   A_2299_SHE20.OutFlagNeg := FALSE;
   A_2299_SHE20.OutpFaultReset := FALSE;
   A_2299_SHE20.OutTrue := FALSE;
   A_2299_SHE20.StFalse := FALSE;
   A_2299_SHE20.StCtoTrue := FALSE;
   A_2299_SHE20.StTrue := FALSE;
   A_2299_SHE20.StCtoFalse := FALSE;
   A_2299_SHE20.StFault := FALSE;
   A_2299_SHE20.OutAlarmNrLog := 0;
   A_2299_SHE20.Par.ParObjectNo := 0;
   A_2299_SHE20.Par.ParMsgType := 0;
   A_2299_SHE20.Par.ParHornCode := 0;
   A_2299_SHE20.Par.ParLogOff := FALSE;
   A_2299_SHE20.Par.spare0401 := FALSE;
   A_2299_SHE20.Par.Par2WorkingCond := FALSE;
   A_2299_SHE20.Par.ParFaultRetry := FALSE;
   A_2299_SHE20.Par.ParBinLevel := FALSE;
   A_2299_SHE20.Par.ParDelayChange := 0;
   A_2299_SHE20.Par.ParDelayTrue := 0;
   A_2299_SHE20.Par.ParDelayFalse := 0;
   A_2299_SHE20.Par.ParTimeoutTrue := 0;
   A_2299_SHE20.Par.ParTimeoutFalse := 0;
   A_2299_SHE20.Par.OutMonTime := 0;
   A_2299_SHE20.Par.OutTransitionTime := 0;
   A_2299_SHE20.Par.OutMonTrue := FALSE;
   A_2299_SHE20.Par.OutMonFalse := FALSE;
   A_2299_SHE20.Par.OutFlagFaultDev := FALSE;
   A_2299_SHE20.Par.OutDelayTime := 0;
   A_2299_SHE21.StCode := 0;
   A_2299_SHE21.InMonTrue := FALSE;
   A_2299_SHE21.InMonFalse := FALSE;
   A_2299_SHE21.InPreAlarmTrue := FALSE;
   A_2299_SHE21.InPreAlarmFalse := FALSE;
   A_2299_SHE21.InStopTrueTime := FALSE;
   A_2299_SHE21.InStopFalseTime := FALSE;
   A_2299_SHE21.InpTrue := FALSE;
   A_2299_SHE21.InpFaultDev := FALSE;
   A_2299_SHE21.CmdRstTrueTime := FALSE;
   A_2299_SHE21.CmdRstFalseTime := FALSE;
   A_2299_SHE21.CmdRunTimeoutTime := FALSE;
   A_2299_SHE21.CmdFaultReset := FALSE;
   A_2299_SHE21.InLocal := FALSE;
   A_2299_SHE21.spare0305 := FALSE;
   A_2299_SHE21.InReport := FALSE;
   A_2299_SHE21.OutTimeoutTime := FALSE;
   A_2299_SHE21.InHWStop := FALSE;
   A_2299_SHE21.InDPFault := FALSE;
   A_2299_SHE21.OutPreAlarmTrue := FALSE;
   A_2299_SHE21.OutPreAlarmFalse := FALSE;
   A_2299_SHE21.OutFlagPos := FALSE;
   A_2299_SHE21.OutFlagNeg := FALSE;
   A_2299_SHE21.OutpFaultReset := FALSE;
   A_2299_SHE21.OutTrue := FALSE;
   A_2299_SHE21.StFalse := FALSE;
   A_2299_SHE21.StCtoTrue := FALSE;
   A_2299_SHE21.StTrue := FALSE;
   A_2299_SHE21.StCtoFalse := FALSE;
   A_2299_SHE21.StFault := FALSE;
   A_2299_SHE21.OutAlarmNrLog := 0;
   A_2299_SHE21.Par.ParObjectNo := 0;
   A_2299_SHE21.Par.ParMsgType := 0;
   A_2299_SHE21.Par.ParHornCode := 0;
   A_2299_SHE21.Par.ParLogOff := FALSE;
   A_2299_SHE21.Par.spare0401 := FALSE;
   A_2299_SHE21.Par.Par2WorkingCond := FALSE;
   A_2299_SHE21.Par.ParFaultRetry := FALSE;
   A_2299_SHE21.Par.ParBinLevel := FALSE;
   A_2299_SHE21.Par.ParDelayChange := 0;
   A_2299_SHE21.Par.ParDelayTrue := 0;
   A_2299_SHE21.Par.ParDelayFalse := 0;
   A_2299_SHE21.Par.ParTimeoutTrue := 0;
   A_2299_SHE21.Par.ParTimeoutFalse := 0;
   A_2299_SHE21.Par.OutMonTime := 0;
   A_2299_SHE21.Par.OutTransitionTime := 0;
   A_2299_SHE21.Par.OutMonTrue := FALSE;
   A_2299_SHE21.Par.OutMonFalse := FALSE;
   A_2299_SHE21.Par.OutFlagFaultDev := FALSE;
   A_2299_SHE21.Par.OutDelayTime := 0;
   A_22_A040Z1.StCode := 0;
   A_22_A040Z1.InMonTrue := FALSE;
   A_22_A040Z1.InMonFalse := FALSE;
   A_22_A040Z1.InPreAlarmTrue := FALSE;
   A_22_A040Z1.InPreAlarmFalse := FALSE;
   A_22_A040Z1.InStopTrueTime := FALSE;
   A_22_A040Z1.InStopFalseTime := FALSE;
   A_22_A040Z1.InpTrue := FALSE;
   A_22_A040Z1.InpFaultDev := FALSE;
   A_22_A040Z1.CmdRstTrueTime := FALSE;
   A_22_A040Z1.CmdRstFalseTime := FALSE;
   A_22_A040Z1.CmdRunTimeoutTime := FALSE;
   A_22_A040Z1.CmdFaultReset := FALSE;
   A_22_A040Z1.InLocal := FALSE;
   A_22_A040Z1.spare0305 := FALSE;
   A_22_A040Z1.InReport := FALSE;
   A_22_A040Z1.OutTimeoutTime := FALSE;
   A_22_A040Z1.InHWStop := FALSE;
   A_22_A040Z1.InDPFault := FALSE;
   A_22_A040Z1.OutPreAlarmTrue := FALSE;
   A_22_A040Z1.OutPreAlarmFalse := FALSE;
   A_22_A040Z1.OutFlagPos := FALSE;
   A_22_A040Z1.OutFlagNeg := FALSE;
   A_22_A040Z1.OutpFaultReset := FALSE;
   A_22_A040Z1.OutTrue := FALSE;
   A_22_A040Z1.StFalse := FALSE;
   A_22_A040Z1.StCtoTrue := FALSE;
   A_22_A040Z1.StTrue := FALSE;
   A_22_A040Z1.StCtoFalse := FALSE;
   A_22_A040Z1.StFault := FALSE;
   A_22_A040Z1.OutAlarmNrLog := 0;
   A_22_A040Z1.Par.ParObjectNo := 0;
   A_22_A040Z1.Par.ParMsgType := 0;
   A_22_A040Z1.Par.ParHornCode := 0;
   A_22_A040Z1.Par.ParLogOff := FALSE;
   A_22_A040Z1.Par.spare0401 := FALSE;
   A_22_A040Z1.Par.Par2WorkingCond := FALSE;
   A_22_A040Z1.Par.ParFaultRetry := FALSE;
   A_22_A040Z1.Par.ParBinLevel := FALSE;
   A_22_A040Z1.Par.ParDelayChange := 0;
   A_22_A040Z1.Par.ParDelayTrue := 0;
   A_22_A040Z1.Par.ParDelayFalse := 0;
   A_22_A040Z1.Par.ParTimeoutTrue := 0;
   A_22_A040Z1.Par.ParTimeoutFalse := 0;
   A_22_A040Z1.Par.OutMonTime := 0;
   A_22_A040Z1.Par.OutTransitionTime := 0;
   A_22_A040Z1.Par.OutMonTrue := FALSE;
   A_22_A040Z1.Par.OutMonFalse := FALSE;
   A_22_A040Z1.Par.OutFlagFaultDev := FALSE;
   A_22_A040Z1.Par.OutDelayTime := 0;
   A_22_A097Z1.StCode := 0;
   A_22_A097Z1.InMonTrue := FALSE;
   A_22_A097Z1.InMonFalse := FALSE;
   A_22_A097Z1.InPreAlarmTrue := FALSE;
   A_22_A097Z1.InPreAlarmFalse := FALSE;
   A_22_A097Z1.InStopTrueTime := FALSE;
   A_22_A097Z1.InStopFalseTime := FALSE;
   A_22_A097Z1.InpTrue := FALSE;
   A_22_A097Z1.InpFaultDev := FALSE;
   A_22_A097Z1.CmdRstTrueTime := FALSE;
   A_22_A097Z1.CmdRstFalseTime := FALSE;
   A_22_A097Z1.CmdRunTimeoutTime := FALSE;
   A_22_A097Z1.CmdFaultReset := FALSE;
   A_22_A097Z1.InLocal := FALSE;
   A_22_A097Z1.spare0305 := FALSE;
   A_22_A097Z1.InReport := FALSE;
   A_22_A097Z1.OutTimeoutTime := FALSE;
   A_22_A097Z1.InHWStop := FALSE;
   A_22_A097Z1.InDPFault := FALSE;
   A_22_A097Z1.OutPreAlarmTrue := FALSE;
   A_22_A097Z1.OutPreAlarmFalse := FALSE;
   A_22_A097Z1.OutFlagPos := FALSE;
   A_22_A097Z1.OutFlagNeg := FALSE;
   A_22_A097Z1.OutpFaultReset := FALSE;
   A_22_A097Z1.OutTrue := FALSE;
   A_22_A097Z1.StFalse := FALSE;
   A_22_A097Z1.StCtoTrue := FALSE;
   A_22_A097Z1.StTrue := FALSE;
   A_22_A097Z1.StCtoFalse := FALSE;
   A_22_A097Z1.StFault := FALSE;
   A_22_A097Z1.OutAlarmNrLog := 0;
   A_22_A097Z1.Par.ParObjectNo := 0;
   A_22_A097Z1.Par.ParMsgType := 0;
   A_22_A097Z1.Par.ParHornCode := 0;
   A_22_A097Z1.Par.ParLogOff := FALSE;
   A_22_A097Z1.Par.spare0401 := FALSE;
   A_22_A097Z1.Par.Par2WorkingCond := FALSE;
   A_22_A097Z1.Par.ParFaultRetry := FALSE;
   A_22_A097Z1.Par.ParBinLevel := FALSE;
   A_22_A097Z1.Par.ParDelayChange := 0;
   A_22_A097Z1.Par.ParDelayTrue := 0;
   A_22_A097Z1.Par.ParDelayFalse := 0;
   A_22_A097Z1.Par.ParTimeoutTrue := 0;
   A_22_A097Z1.Par.ParTimeoutFalse := 0;
   A_22_A097Z1.Par.OutMonTime := 0;
   A_22_A097Z1.Par.OutTransitionTime := 0;
   A_22_A097Z1.Par.OutMonTrue := FALSE;
   A_22_A097Z1.Par.OutMonFalse := FALSE;
   A_22_A097Z1.Par.OutFlagFaultDev := FALSE;
   A_22_A097Z1.Par.OutDelayTime := 0;
   A_22_A098Z1.StCode := 0;
   A_22_A098Z1.InMonTrue := FALSE;
   A_22_A098Z1.InMonFalse := FALSE;
   A_22_A098Z1.InPreAlarmTrue := FALSE;
   A_22_A098Z1.InPreAlarmFalse := FALSE;
   A_22_A098Z1.InStopTrueTime := FALSE;
   A_22_A098Z1.InStopFalseTime := FALSE;
   A_22_A098Z1.InpTrue := FALSE;
   A_22_A098Z1.InpFaultDev := FALSE;
   A_22_A098Z1.CmdRstTrueTime := FALSE;
   A_22_A098Z1.CmdRstFalseTime := FALSE;
   A_22_A098Z1.CmdRunTimeoutTime := FALSE;
   A_22_A098Z1.CmdFaultReset := FALSE;
   A_22_A098Z1.InLocal := FALSE;
   A_22_A098Z1.spare0305 := FALSE;
   A_22_A098Z1.InReport := FALSE;
   A_22_A098Z1.OutTimeoutTime := FALSE;
   A_22_A098Z1.InHWStop := FALSE;
   A_22_A098Z1.InDPFault := FALSE;
   A_22_A098Z1.OutPreAlarmTrue := FALSE;
   A_22_A098Z1.OutPreAlarmFalse := FALSE;
   A_22_A098Z1.OutFlagPos := FALSE;
   A_22_A098Z1.OutFlagNeg := FALSE;
   A_22_A098Z1.OutpFaultReset := FALSE;
   A_22_A098Z1.OutTrue := FALSE;
   A_22_A098Z1.StFalse := FALSE;
   A_22_A098Z1.StCtoTrue := FALSE;
   A_22_A098Z1.StTrue := FALSE;
   A_22_A098Z1.StCtoFalse := FALSE;
   A_22_A098Z1.StFault := FALSE;
   A_22_A098Z1.OutAlarmNrLog := 0;
   A_22_A098Z1.Par.ParObjectNo := 0;
   A_22_A098Z1.Par.ParMsgType := 0;
   A_22_A098Z1.Par.ParHornCode := 0;
   A_22_A098Z1.Par.ParLogOff := FALSE;
   A_22_A098Z1.Par.spare0401 := FALSE;
   A_22_A098Z1.Par.Par2WorkingCond := FALSE;
   A_22_A098Z1.Par.ParFaultRetry := FALSE;
   A_22_A098Z1.Par.ParBinLevel := FALSE;
   A_22_A098Z1.Par.ParDelayChange := 0;
   A_22_A098Z1.Par.ParDelayTrue := 0;
   A_22_A098Z1.Par.ParDelayFalse := 0;
   A_22_A098Z1.Par.ParTimeoutTrue := 0;
   A_22_A098Z1.Par.ParTimeoutFalse := 0;
   A_22_A098Z1.Par.OutMonTime := 0;
   A_22_A098Z1.Par.OutTransitionTime := 0;
   A_22_A098Z1.Par.OutMonTrue := FALSE;
   A_22_A098Z1.Par.OutMonFalse := FALSE;
   A_22_A098Z1.Par.OutFlagFaultDev := FALSE;
   A_22_A098Z1.Par.OutDelayTime := 0;
   A_22_K091Z1.StCode := 0;
   A_22_K091Z1.InMonTrue := FALSE;
   A_22_K091Z1.InMonFalse := FALSE;
   A_22_K091Z1.InPreAlarmTrue := FALSE;
   A_22_K091Z1.InPreAlarmFalse := FALSE;
   A_22_K091Z1.InStopTrueTime := FALSE;
   A_22_K091Z1.InStopFalseTime := FALSE;
   A_22_K091Z1.InpTrue := FALSE;
   A_22_K091Z1.InpFaultDev := FALSE;
   A_22_K091Z1.CmdRstTrueTime := FALSE;
   A_22_K091Z1.CmdRstFalseTime := FALSE;
   A_22_K091Z1.CmdRunTimeoutTime := FALSE;
   A_22_K091Z1.CmdFaultReset := FALSE;
   A_22_K091Z1.InLocal := FALSE;
   A_22_K091Z1.spare0305 := FALSE;
   A_22_K091Z1.InReport := FALSE;
   A_22_K091Z1.OutTimeoutTime := FALSE;
   A_22_K091Z1.InHWStop := FALSE;
   A_22_K091Z1.InDPFault := FALSE;
   A_22_K091Z1.OutPreAlarmTrue := FALSE;
   A_22_K091Z1.OutPreAlarmFalse := FALSE;
   A_22_K091Z1.OutFlagPos := FALSE;
   A_22_K091Z1.OutFlagNeg := FALSE;
   A_22_K091Z1.OutpFaultReset := FALSE;
   A_22_K091Z1.OutTrue := FALSE;
   A_22_K091Z1.StFalse := FALSE;
   A_22_K091Z1.StCtoTrue := FALSE;
   A_22_K091Z1.StTrue := FALSE;
   A_22_K091Z1.StCtoFalse := FALSE;
   A_22_K091Z1.StFault := FALSE;
   A_22_K091Z1.OutAlarmNrLog := 0;
   A_22_K091Z1.Par.ParObjectNo := 0;
   A_22_K091Z1.Par.ParMsgType := 0;
   A_22_K091Z1.Par.ParHornCode := 0;
   A_22_K091Z1.Par.ParLogOff := FALSE;
   A_22_K091Z1.Par.spare0401 := FALSE;
   A_22_K091Z1.Par.Par2WorkingCond := FALSE;
   A_22_K091Z1.Par.ParFaultRetry := FALSE;
   A_22_K091Z1.Par.ParBinLevel := FALSE;
   A_22_K091Z1.Par.ParDelayChange := 0;
   A_22_K091Z1.Par.ParDelayTrue := 0;
   A_22_K091Z1.Par.ParDelayFalse := 0;
   A_22_K091Z1.Par.ParTimeoutTrue := 0;
   A_22_K091Z1.Par.ParTimeoutFalse := 0;
   A_22_K091Z1.Par.OutMonTime := 0;
   A_22_K091Z1.Par.OutTransitionTime := 0;
   A_22_K091Z1.Par.OutMonTrue := FALSE;
   A_22_K091Z1.Par.OutMonFalse := FALSE;
   A_22_K091Z1.Par.OutFlagFaultDev := FALSE;
   A_22_K091Z1.Par.OutDelayTime := 0;
   A_22_K738R1.StCode := 0;
   A_22_K738R1.InMonTrue := FALSE;
   A_22_K738R1.InMonFalse := FALSE;
   A_22_K738R1.InPreAlarmTrue := FALSE;
   A_22_K738R1.InPreAlarmFalse := FALSE;
   A_22_K738R1.InStopTrueTime := FALSE;
   A_22_K738R1.InStopFalseTime := FALSE;
   A_22_K738R1.InpTrue := FALSE;
   A_22_K738R1.InpFaultDev := FALSE;
   A_22_K738R1.CmdRstTrueTime := FALSE;
   A_22_K738R1.CmdRstFalseTime := FALSE;
   A_22_K738R1.CmdRunTimeoutTime := FALSE;
   A_22_K738R1.CmdFaultReset := FALSE;
   A_22_K738R1.InLocal := FALSE;
   A_22_K738R1.spare0305 := FALSE;
   A_22_K738R1.InReport := FALSE;
   A_22_K738R1.OutTimeoutTime := FALSE;
   A_22_K738R1.InHWStop := FALSE;
   A_22_K738R1.InDPFault := FALSE;
   A_22_K738R1.OutPreAlarmTrue := FALSE;
   A_22_K738R1.OutPreAlarmFalse := FALSE;
   A_22_K738R1.OutFlagPos := FALSE;
   A_22_K738R1.OutFlagNeg := FALSE;
   A_22_K738R1.OutpFaultReset := FALSE;
   A_22_K738R1.OutTrue := FALSE;
   A_22_K738R1.StFalse := FALSE;
   A_22_K738R1.StCtoTrue := FALSE;
   A_22_K738R1.StTrue := FALSE;
   A_22_K738R1.StCtoFalse := FALSE;
   A_22_K738R1.StFault := FALSE;
   A_22_K738R1.OutAlarmNrLog := 0;
   A_22_K738R1.Par.ParObjectNo := 0;
   A_22_K738R1.Par.ParMsgType := 0;
   A_22_K738R1.Par.ParHornCode := 0;
   A_22_K738R1.Par.ParLogOff := FALSE;
   A_22_K738R1.Par.spare0401 := FALSE;
   A_22_K738R1.Par.Par2WorkingCond := FALSE;
   A_22_K738R1.Par.ParFaultRetry := FALSE;
   A_22_K738R1.Par.ParBinLevel := FALSE;
   A_22_K738R1.Par.ParDelayChange := 0;
   A_22_K738R1.Par.ParDelayTrue := 0;
   A_22_K738R1.Par.ParDelayFalse := 0;
   A_22_K738R1.Par.ParTimeoutTrue := 0;
   A_22_K738R1.Par.ParTimeoutFalse := 0;
   A_22_K738R1.Par.OutMonTime := 0;
   A_22_K738R1.Par.OutTransitionTime := 0;
   A_22_K738R1.Par.OutMonTrue := FALSE;
   A_22_K738R1.Par.OutMonFalse := FALSE;
   A_22_K738R1.Par.OutFlagFaultDev := FALSE;
   A_22_K738R1.Par.OutDelayTime := 0;
   A_22_K838R1.StCode := 0;
   A_22_K838R1.InMonTrue := FALSE;
   A_22_K838R1.InMonFalse := FALSE;
   A_22_K838R1.InPreAlarmTrue := FALSE;
   A_22_K838R1.InPreAlarmFalse := FALSE;
   A_22_K838R1.InStopTrueTime := FALSE;
   A_22_K838R1.InStopFalseTime := FALSE;
   A_22_K838R1.InpTrue := FALSE;
   A_22_K838R1.InpFaultDev := FALSE;
   A_22_K838R1.CmdRstTrueTime := FALSE;
   A_22_K838R1.CmdRstFalseTime := FALSE;
   A_22_K838R1.CmdRunTimeoutTime := FALSE;
   A_22_K838R1.CmdFaultReset := FALSE;
   A_22_K838R1.InLocal := FALSE;
   A_22_K838R1.spare0305 := FALSE;
   A_22_K838R1.InReport := FALSE;
   A_22_K838R1.OutTimeoutTime := FALSE;
   A_22_K838R1.InHWStop := FALSE;
   A_22_K838R1.InDPFault := FALSE;
   A_22_K838R1.OutPreAlarmTrue := FALSE;
   A_22_K838R1.OutPreAlarmFalse := FALSE;
   A_22_K838R1.OutFlagPos := FALSE;
   A_22_K838R1.OutFlagNeg := FALSE;
   A_22_K838R1.OutpFaultReset := FALSE;
   A_22_K838R1.OutTrue := FALSE;
   A_22_K838R1.StFalse := FALSE;
   A_22_K838R1.StCtoTrue := FALSE;
   A_22_K838R1.StTrue := FALSE;
   A_22_K838R1.StCtoFalse := FALSE;
   A_22_K838R1.StFault := FALSE;
   A_22_K838R1.OutAlarmNrLog := 0;
   A_22_K838R1.Par.ParObjectNo := 0;
   A_22_K838R1.Par.ParMsgType := 0;
   A_22_K838R1.Par.ParHornCode := 0;
   A_22_K838R1.Par.ParLogOff := FALSE;
   A_22_K838R1.Par.spare0401 := FALSE;
   A_22_K838R1.Par.Par2WorkingCond := FALSE;
   A_22_K838R1.Par.ParFaultRetry := FALSE;
   A_22_K838R1.Par.ParBinLevel := FALSE;
   A_22_K838R1.Par.ParDelayChange := 0;
   A_22_K838R1.Par.ParDelayTrue := 0;
   A_22_K838R1.Par.ParDelayFalse := 0;
   A_22_K838R1.Par.ParTimeoutTrue := 0;
   A_22_K838R1.Par.ParTimeoutFalse := 0;
   A_22_K838R1.Par.OutMonTime := 0;
   A_22_K838R1.Par.OutTransitionTime := 0;
   A_22_K838R1.Par.OutMonTrue := FALSE;
   A_22_K838R1.Par.OutMonFalse := FALSE;
   A_22_K838R1.Par.OutFlagFaultDev := FALSE;
   A_22_K838R1.Par.OutDelayTime := 0;
   A_22_Q390Z1.StCode := 0;
   A_22_Q390Z1.InMonTrue := FALSE;
   A_22_Q390Z1.InMonFalse := FALSE;
   A_22_Q390Z1.InPreAlarmTrue := FALSE;
   A_22_Q390Z1.InPreAlarmFalse := FALSE;
   A_22_Q390Z1.InStopTrueTime := FALSE;
   A_22_Q390Z1.InStopFalseTime := FALSE;
   A_22_Q390Z1.InpTrue := FALSE;
   A_22_Q390Z1.InpFaultDev := FALSE;
   A_22_Q390Z1.CmdRstTrueTime := FALSE;
   A_22_Q390Z1.CmdRstFalseTime := FALSE;
   A_22_Q390Z1.CmdRunTimeoutTime := FALSE;
   A_22_Q390Z1.CmdFaultReset := FALSE;
   A_22_Q390Z1.InLocal := FALSE;
   A_22_Q390Z1.spare0305 := FALSE;
   A_22_Q390Z1.InReport := FALSE;
   A_22_Q390Z1.OutTimeoutTime := FALSE;
   A_22_Q390Z1.InHWStop := FALSE;
   A_22_Q390Z1.InDPFault := FALSE;
   A_22_Q390Z1.OutPreAlarmTrue := FALSE;
   A_22_Q390Z1.OutPreAlarmFalse := FALSE;
   A_22_Q390Z1.OutFlagPos := FALSE;
   A_22_Q390Z1.OutFlagNeg := FALSE;
   A_22_Q390Z1.OutpFaultReset := FALSE;
   A_22_Q390Z1.OutTrue := FALSE;
   A_22_Q390Z1.StFalse := FALSE;
   A_22_Q390Z1.StCtoTrue := FALSE;
   A_22_Q390Z1.StTrue := FALSE;
   A_22_Q390Z1.StCtoFalse := FALSE;
   A_22_Q390Z1.StFault := FALSE;
   A_22_Q390Z1.OutAlarmNrLog := 0;
   A_22_Q390Z1.Par.ParObjectNo := 0;
   A_22_Q390Z1.Par.ParMsgType := 0;
   A_22_Q390Z1.Par.ParHornCode := 0;
   A_22_Q390Z1.Par.ParLogOff := FALSE;
   A_22_Q390Z1.Par.spare0401 := FALSE;
   A_22_Q390Z1.Par.Par2WorkingCond := FALSE;
   A_22_Q390Z1.Par.ParFaultRetry := FALSE;
   A_22_Q390Z1.Par.ParBinLevel := FALSE;
   A_22_Q390Z1.Par.ParDelayChange := 0;
   A_22_Q390Z1.Par.ParDelayTrue := 0;
   A_22_Q390Z1.Par.ParDelayFalse := 0;
   A_22_Q390Z1.Par.ParTimeoutTrue := 0;
   A_22_Q390Z1.Par.ParTimeoutFalse := 0;
   A_22_Q390Z1.Par.OutMonTime := 0;
   A_22_Q390Z1.Par.OutTransitionTime := 0;
   A_22_Q390Z1.Par.OutMonTrue := FALSE;
   A_22_Q390Z1.Par.OutMonFalse := FALSE;
   A_22_Q390Z1.Par.OutFlagFaultDev := FALSE;
   A_22_Q390Z1.Par.OutDelayTime := 0;
   A_22_Q445Z1.StCode := 0;
   A_22_Q445Z1.InMonTrue := FALSE;
   A_22_Q445Z1.InMonFalse := FALSE;
   A_22_Q445Z1.InPreAlarmTrue := FALSE;
   A_22_Q445Z1.InPreAlarmFalse := FALSE;
   A_22_Q445Z1.InStopTrueTime := FALSE;
   A_22_Q445Z1.InStopFalseTime := FALSE;
   A_22_Q445Z1.InpTrue := FALSE;
   A_22_Q445Z1.InpFaultDev := FALSE;
   A_22_Q445Z1.CmdRstTrueTime := FALSE;
   A_22_Q445Z1.CmdRstFalseTime := FALSE;
   A_22_Q445Z1.CmdRunTimeoutTime := FALSE;
   A_22_Q445Z1.CmdFaultReset := FALSE;
   A_22_Q445Z1.InLocal := FALSE;
   A_22_Q445Z1.spare0305 := FALSE;
   A_22_Q445Z1.InReport := FALSE;
   A_22_Q445Z1.OutTimeoutTime := FALSE;
   A_22_Q445Z1.InHWStop := FALSE;
   A_22_Q445Z1.InDPFault := FALSE;
   A_22_Q445Z1.OutPreAlarmTrue := FALSE;
   A_22_Q445Z1.OutPreAlarmFalse := FALSE;
   A_22_Q445Z1.OutFlagPos := FALSE;
   A_22_Q445Z1.OutFlagNeg := FALSE;
   A_22_Q445Z1.OutpFaultReset := FALSE;
   A_22_Q445Z1.OutTrue := FALSE;
   A_22_Q445Z1.StFalse := FALSE;
   A_22_Q445Z1.StCtoTrue := FALSE;
   A_22_Q445Z1.StTrue := FALSE;
   A_22_Q445Z1.StCtoFalse := FALSE;
   A_22_Q445Z1.StFault := FALSE;
   A_22_Q445Z1.OutAlarmNrLog := 0;
   A_22_Q445Z1.Par.ParObjectNo := 0;
   A_22_Q445Z1.Par.ParMsgType := 0;
   A_22_Q445Z1.Par.ParHornCode := 0;
   A_22_Q445Z1.Par.ParLogOff := FALSE;
   A_22_Q445Z1.Par.spare0401 := FALSE;
   A_22_Q445Z1.Par.Par2WorkingCond := FALSE;
   A_22_Q445Z1.Par.ParFaultRetry := FALSE;
   A_22_Q445Z1.Par.ParBinLevel := FALSE;
   A_22_Q445Z1.Par.ParDelayChange := 0;
   A_22_Q445Z1.Par.ParDelayTrue := 0;
   A_22_Q445Z1.Par.ParDelayFalse := 0;
   A_22_Q445Z1.Par.ParTimeoutTrue := 0;
   A_22_Q445Z1.Par.ParTimeoutFalse := 0;
   A_22_Q445Z1.Par.OutMonTime := 0;
   A_22_Q445Z1.Par.OutTransitionTime := 0;
   A_22_Q445Z1.Par.OutMonTrue := FALSE;
   A_22_Q445Z1.Par.OutMonFalse := FALSE;
   A_22_Q445Z1.Par.OutFlagFaultDev := FALSE;
   A_22_Q445Z1.Par.OutDelayTime := 0;
   A_22_S_H097Z1.StCode := 0;
   A_22_S_H097Z1.InMonTrue := FALSE;
   A_22_S_H097Z1.InMonFalse := FALSE;
   A_22_S_H097Z1.InPreAlarmTrue := FALSE;
   A_22_S_H097Z1.InPreAlarmFalse := FALSE;
   A_22_S_H097Z1.InStopTrueTime := FALSE;
   A_22_S_H097Z1.InStopFalseTime := FALSE;
   A_22_S_H097Z1.InpTrue := FALSE;
   A_22_S_H097Z1.InpFaultDev := FALSE;
   A_22_S_H097Z1.CmdRstTrueTime := FALSE;
   A_22_S_H097Z1.CmdRstFalseTime := FALSE;
   A_22_S_H097Z1.CmdRunTimeoutTime := FALSE;
   A_22_S_H097Z1.CmdFaultReset := FALSE;
   A_22_S_H097Z1.InLocal := FALSE;
   A_22_S_H097Z1.spare0305 := FALSE;
   A_22_S_H097Z1.InReport := FALSE;
   A_22_S_H097Z1.OutTimeoutTime := FALSE;
   A_22_S_H097Z1.InHWStop := FALSE;
   A_22_S_H097Z1.InDPFault := FALSE;
   A_22_S_H097Z1.OutPreAlarmTrue := FALSE;
   A_22_S_H097Z1.OutPreAlarmFalse := FALSE;
   A_22_S_H097Z1.OutFlagPos := FALSE;
   A_22_S_H097Z1.OutFlagNeg := FALSE;
   A_22_S_H097Z1.OutpFaultReset := FALSE;
   A_22_S_H097Z1.OutTrue := FALSE;
   A_22_S_H097Z1.StFalse := FALSE;
   A_22_S_H097Z1.StCtoTrue := FALSE;
   A_22_S_H097Z1.StTrue := FALSE;
   A_22_S_H097Z1.StCtoFalse := FALSE;
   A_22_S_H097Z1.StFault := FALSE;
   A_22_S_H097Z1.OutAlarmNrLog := 0;
   A_22_S_H097Z1.Par.ParObjectNo := 0;
   A_22_S_H097Z1.Par.ParMsgType := 0;
   A_22_S_H097Z1.Par.ParHornCode := 0;
   A_22_S_H097Z1.Par.ParLogOff := FALSE;
   A_22_S_H097Z1.Par.spare0401 := FALSE;
   A_22_S_H097Z1.Par.Par2WorkingCond := FALSE;
   A_22_S_H097Z1.Par.ParFaultRetry := FALSE;
   A_22_S_H097Z1.Par.ParBinLevel := FALSE;
   A_22_S_H097Z1.Par.ParDelayChange := 0;
   A_22_S_H097Z1.Par.ParDelayTrue := 0;
   A_22_S_H097Z1.Par.ParDelayFalse := 0;
   A_22_S_H097Z1.Par.ParTimeoutTrue := 0;
   A_22_S_H097Z1.Par.ParTimeoutFalse := 0;
   A_22_S_H097Z1.Par.OutMonTime := 0;
   A_22_S_H097Z1.Par.OutTransitionTime := 0;
   A_22_S_H097Z1.Par.OutMonTrue := FALSE;
   A_22_S_H097Z1.Par.OutMonFalse := FALSE;
   A_22_S_H097Z1.Par.OutFlagFaultDev := FALSE;
   A_22_S_H097Z1.Par.OutDelayTime := 0;
   A_22_A458Z1.StCode := 0;
   A_22_A458Z1.InMonTrue := FALSE;
   A_22_A458Z1.InMonFalse := FALSE;
   A_22_A458Z1.InPreAlarmTrue := FALSE;
   A_22_A458Z1.InPreAlarmFalse := FALSE;
   A_22_A458Z1.InStopTrueTime := FALSE;
   A_22_A458Z1.InStopFalseTime := FALSE;
   A_22_A458Z1.InpTrue := FALSE;
   A_22_A458Z1.InpFaultDev := FALSE;
   A_22_A458Z1.CmdRstTrueTime := FALSE;
   A_22_A458Z1.CmdRstFalseTime := FALSE;
   A_22_A458Z1.CmdRunTimeoutTime := FALSE;
   A_22_A458Z1.CmdFaultReset := FALSE;
   A_22_A458Z1.InLocal := FALSE;
   A_22_A458Z1.spare0305 := FALSE;
   A_22_A458Z1.InReport := FALSE;
   A_22_A458Z1.OutTimeoutTime := FALSE;
   A_22_A458Z1.InHWStop := FALSE;
   A_22_A458Z1.InDPFault := FALSE;
   A_22_A458Z1.OutPreAlarmTrue := FALSE;
   A_22_A458Z1.OutPreAlarmFalse := FALSE;
   A_22_A458Z1.OutFlagPos := FALSE;
   A_22_A458Z1.OutFlagNeg := FALSE;
   A_22_A458Z1.OutpFaultReset := FALSE;
   A_22_A458Z1.OutTrue := FALSE;
   A_22_A458Z1.StFalse := FALSE;
   A_22_A458Z1.StCtoTrue := FALSE;
   A_22_A458Z1.StTrue := FALSE;
   A_22_A458Z1.StCtoFalse := FALSE;
   A_22_A458Z1.StFault := FALSE;
   A_22_A458Z1.OutAlarmNrLog := 0;
   A_22_A458Z1.Par.ParObjectNo := 0;
   A_22_A458Z1.Par.ParMsgType := 0;
   A_22_A458Z1.Par.ParHornCode := 0;
   A_22_A458Z1.Par.ParLogOff := FALSE;
   A_22_A458Z1.Par.spare0401 := FALSE;
   A_22_A458Z1.Par.Par2WorkingCond := FALSE;
   A_22_A458Z1.Par.ParFaultRetry := FALSE;
   A_22_A458Z1.Par.ParBinLevel := FALSE;
   A_22_A458Z1.Par.ParDelayChange := 0;
   A_22_A458Z1.Par.ParDelayTrue := 0;
   A_22_A458Z1.Par.ParDelayFalse := 0;
   A_22_A458Z1.Par.ParTimeoutTrue := 0;
   A_22_A458Z1.Par.ParTimeoutFalse := 0;
   A_22_A458Z1.Par.OutMonTime := 0;
   A_22_A458Z1.Par.OutTransitionTime := 0;
   A_22_A458Z1.Par.OutMonTrue := FALSE;
   A_22_A458Z1.Par.OutMonFalse := FALSE;
   A_22_A458Z1.Par.OutFlagFaultDev := FALSE;
   A_22_A458Z1.Par.OutDelayTime := 0;
   A_22_D1B065.StCode := 0;
   A_22_D1B065.InMonTrue := FALSE;
   A_22_D1B065.InMonFalse := FALSE;
   A_22_D1B065.InPreAlarmTrue := FALSE;
   A_22_D1B065.InPreAlarmFalse := FALSE;
   A_22_D1B065.InStopTrueTime := FALSE;
   A_22_D1B065.InStopFalseTime := FALSE;
   A_22_D1B065.InpTrue := FALSE;
   A_22_D1B065.InpFaultDev := FALSE;
   A_22_D1B065.CmdRstTrueTime := FALSE;
   A_22_D1B065.CmdRstFalseTime := FALSE;
   A_22_D1B065.CmdRunTimeoutTime := FALSE;
   A_22_D1B065.CmdFaultReset := FALSE;
   A_22_D1B065.InLocal := FALSE;
   A_22_D1B065.spare0305 := FALSE;
   A_22_D1B065.InReport := FALSE;
   A_22_D1B065.OutTimeoutTime := FALSE;
   A_22_D1B065.InHWStop := FALSE;
   A_22_D1B065.InDPFault := FALSE;
   A_22_D1B065.OutPreAlarmTrue := FALSE;
   A_22_D1B065.OutPreAlarmFalse := FALSE;
   A_22_D1B065.OutFlagPos := FALSE;
   A_22_D1B065.OutFlagNeg := FALSE;
   A_22_D1B065.OutpFaultReset := FALSE;
   A_22_D1B065.OutTrue := FALSE;
   A_22_D1B065.StFalse := FALSE;
   A_22_D1B065.StCtoTrue := FALSE;
   A_22_D1B065.StTrue := FALSE;
   A_22_D1B065.StCtoFalse := FALSE;
   A_22_D1B065.StFault := FALSE;
   A_22_D1B065.OutAlarmNrLog := 0;
   A_22_D1B065.Par.ParObjectNo := 0;
   A_22_D1B065.Par.ParMsgType := 0;
   A_22_D1B065.Par.ParHornCode := 0;
   A_22_D1B065.Par.ParLogOff := FALSE;
   A_22_D1B065.Par.spare0401 := FALSE;
   A_22_D1B065.Par.Par2WorkingCond := FALSE;
   A_22_D1B065.Par.ParFaultRetry := FALSE;
   A_22_D1B065.Par.ParBinLevel := FALSE;
   A_22_D1B065.Par.ParDelayChange := 0;
   A_22_D1B065.Par.ParDelayTrue := 0;
   A_22_D1B065.Par.ParDelayFalse := 0;
   A_22_D1B065.Par.ParTimeoutTrue := 0;
   A_22_D1B065.Par.ParTimeoutFalse := 0;
   A_22_D1B065.Par.OutMonTime := 0;
   A_22_D1B065.Par.OutTransitionTime := 0;
   A_22_D1B065.Par.OutMonTrue := FALSE;
   A_22_D1B065.Par.OutMonFalse := FALSE;
   A_22_D1B065.Par.OutFlagFaultDev := FALSE;
   A_22_D1B065.Par.OutDelayTime := 0;
   A_22_A408Z1I1.StCode := 0;
   A_22_A408Z1I1.InMonTrue := FALSE;
   A_22_A408Z1I1.InMonFalse := FALSE;
   A_22_A408Z1I1.InPreAlarmTrue := FALSE;
   A_22_A408Z1I1.InPreAlarmFalse := FALSE;
   A_22_A408Z1I1.InStopTrueTime := FALSE;
   A_22_A408Z1I1.InStopFalseTime := FALSE;
   A_22_A408Z1I1.InpTrue := FALSE;
   A_22_A408Z1I1.InpFaultDev := FALSE;
   A_22_A408Z1I1.CmdRstTrueTime := FALSE;
   A_22_A408Z1I1.CmdRstFalseTime := FALSE;
   A_22_A408Z1I1.CmdRunTimeoutTime := FALSE;
   A_22_A408Z1I1.CmdFaultReset := FALSE;
   A_22_A408Z1I1.InLocal := FALSE;
   A_22_A408Z1I1.spare0305 := FALSE;
   A_22_A408Z1I1.InReport := FALSE;
   A_22_A408Z1I1.OutTimeoutTime := FALSE;
   A_22_A408Z1I1.InHWStop := FALSE;
   A_22_A408Z1I1.InDPFault := FALSE;
   A_22_A408Z1I1.OutPreAlarmTrue := FALSE;
   A_22_A408Z1I1.OutPreAlarmFalse := FALSE;
   A_22_A408Z1I1.OutFlagPos := FALSE;
   A_22_A408Z1I1.OutFlagNeg := FALSE;
   A_22_A408Z1I1.OutpFaultReset := FALSE;
   A_22_A408Z1I1.OutTrue := FALSE;
   A_22_A408Z1I1.StFalse := FALSE;
   A_22_A408Z1I1.StCtoTrue := FALSE;
   A_22_A408Z1I1.StTrue := FALSE;
   A_22_A408Z1I1.StCtoFalse := FALSE;
   A_22_A408Z1I1.StFault := FALSE;
   A_22_A408Z1I1.OutAlarmNrLog := 0;
   A_22_A408Z1I1.Par.ParObjectNo := 0;
   A_22_A408Z1I1.Par.ParMsgType := 0;
   A_22_A408Z1I1.Par.ParHornCode := 0;
   A_22_A408Z1I1.Par.ParLogOff := FALSE;
   A_22_A408Z1I1.Par.spare0401 := FALSE;
   A_22_A408Z1I1.Par.Par2WorkingCond := FALSE;
   A_22_A408Z1I1.Par.ParFaultRetry := FALSE;
   A_22_A408Z1I1.Par.ParBinLevel := FALSE;
   A_22_A408Z1I1.Par.ParDelayChange := 0;
   A_22_A408Z1I1.Par.ParDelayTrue := 0;
   A_22_A408Z1I1.Par.ParDelayFalse := 0;
   A_22_A408Z1I1.Par.ParTimeoutTrue := 0;
   A_22_A408Z1I1.Par.ParTimeoutFalse := 0;
   A_22_A408Z1I1.Par.OutMonTime := 0;
   A_22_A408Z1I1.Par.OutTransitionTime := 0;
   A_22_A408Z1I1.Par.OutMonTrue := FALSE;
   A_22_A408Z1I1.Par.OutMonFalse := FALSE;
   A_22_A408Z1I1.Par.OutFlagFaultDev := FALSE;
   A_22_A408Z1I1.Par.OutDelayTime := 0;
   A_22_A408Z1O1.StCode := 0;
   A_22_A408Z1O1.InEnable := FALSE;
   A_22_A408Z1O1.spare0201 := FALSE;
   A_22_A408Z1O1.InContinuous := FALSE;
   A_22_A408Z1O1.spare0203 := FALSE;
   A_22_A408Z1O1.spare0204 := FALSE;
   A_22_A408Z1O1.spare0205 := FALSE;
   A_22_A408Z1O1.InpRun := FALSE;
   A_22_A408Z1O1.InpFaultDev := FALSE;
   A_22_A408Z1O1.CmdOff := FALSE;
   A_22_A408Z1O1.CmdOn := FALSE;
   A_22_A408Z1O1.CmdNext := FALSE;
   A_22_A408Z1O1.CmdFaultReset := FALSE;
   A_22_A408Z1O1.InLocal := FALSE;
   A_22_A408Z1O1.InManual := FALSE;
   A_22_A408Z1O1.InReport := FALSE;
   A_22_A408Z1O1.InSeqStop := FALSE;
   A_22_A408Z1O1.InHWStop := FALSE;
   A_22_A408Z1O1.InDPFault := FALSE;
   A_22_A408Z1O1.OutIdling := FALSE;
   A_22_A408Z1O1.OutWarning := FALSE;
   A_22_A408Z1O1.spare0404 := FALSE;
   A_22_A408Z1O1.spare0405 := FALSE;
   A_22_A408Z1O1.OutpFaultReset := FALSE;
   A_22_A408Z1O1.OutpRun := FALSE;
   A_22_A408Z1O1.StStopped := FALSE;
   A_22_A408Z1O1.StStarting := FALSE;
   A_22_A408Z1O1.StStarted := FALSE;
   A_22_A408Z1O1.spare0503 := FALSE;
   A_22_A408Z1O1.StFault := FALSE;
   A_22_A408Z1O1.StFalse := FALSE;
   A_22_A408Z1O1.spare0506 := FALSE;
   A_22_A408Z1O1.OutPausing := FALSE;
   A_22_A408Z1O1.OutAlarmNrLog := 0;
   A_22_A408Z1O1.Par.ParObjectNo := 0;
   A_22_A408Z1O1.Par.ParMsgType := 0;
   A_22_A408Z1O1.Par.ParHornCode := 0;
   A_22_A408Z1O1.Par.ParLogOff := FALSE;
   A_22_A408Z1O1.Par.ParManual := FALSE;
   A_22_A408Z1O1.Par.ParContinuous := FALSE;
   A_22_A408Z1O1.Par.ParPulse := FALSE;
   A_22_A408Z1O1.Par.ParPulsing := FALSE;
   A_22_A408Z1O1.Par.ParFilter := FALSE;
   A_22_A408Z1O1.Par.ParOnTime := 0;
   A_22_A408Z1O1.Par.ParOffTime := 0;
   A_22_A408Z1O1.Par.ParIdlingTime := 0;
   A_22_A408Z1O1.Par.ParDelayTime := 0;
   A_22_A408Z1O1.Par.OutTime := 0;
   A_22_A408Z1O1.Par.OutDelayTime := 0;
   A_22_A408Z1O1.Par.spare26 := 0;
   A_22_A408Z1O1.Par.spare28 := 0;
   A_22_A408Z1O1.Par.InOutManPulseLen := 0;
   A_22_A700Z1.StCode := 0;
   A_22_A700Z1.InMonTrue := FALSE;
   A_22_A700Z1.InMonFalse := FALSE;
   A_22_A700Z1.InPreAlarmTrue := FALSE;
   A_22_A700Z1.InPreAlarmFalse := FALSE;
   A_22_A700Z1.InStopTrueTime := FALSE;
   A_22_A700Z1.InStopFalseTime := FALSE;
   A_22_A700Z1.InpTrue := FALSE;
   A_22_A700Z1.InpFaultDev := FALSE;
   A_22_A700Z1.CmdRstTrueTime := FALSE;
   A_22_A700Z1.CmdRstFalseTime := FALSE;
   A_22_A700Z1.CmdRunTimeoutTime := FALSE;
   A_22_A700Z1.CmdFaultReset := FALSE;
   A_22_A700Z1.InLocal := FALSE;
   A_22_A700Z1.spare0305 := FALSE;
   A_22_A700Z1.InReport := FALSE;
   A_22_A700Z1.OutTimeoutTime := FALSE;
   A_22_A700Z1.InHWStop := FALSE;
   A_22_A700Z1.InDPFault := FALSE;
   A_22_A700Z1.OutPreAlarmTrue := FALSE;
   A_22_A700Z1.OutPreAlarmFalse := FALSE;
   A_22_A700Z1.OutFlagPos := FALSE;
   A_22_A700Z1.OutFlagNeg := FALSE;
   A_22_A700Z1.OutpFaultReset := FALSE;
   A_22_A700Z1.OutTrue := FALSE;
   A_22_A700Z1.StFalse := FALSE;
   A_22_A700Z1.StCtoTrue := FALSE;
   A_22_A700Z1.StTrue := FALSE;
   A_22_A700Z1.StCtoFalse := FALSE;
   A_22_A700Z1.StFault := FALSE;
   A_22_A700Z1.OutAlarmNrLog := 0;
   A_22_A700Z1.Par.ParObjectNo := 0;
   A_22_A700Z1.Par.ParMsgType := 0;
   A_22_A700Z1.Par.ParHornCode := 0;
   A_22_A700Z1.Par.ParLogOff := FALSE;
   A_22_A700Z1.Par.spare0401 := FALSE;
   A_22_A700Z1.Par.Par2WorkingCond := FALSE;
   A_22_A700Z1.Par.ParFaultRetry := FALSE;
   A_22_A700Z1.Par.ParBinLevel := FALSE;
   A_22_A700Z1.Par.ParDelayChange := 0;
   A_22_A700Z1.Par.ParDelayTrue := 0;
   A_22_A700Z1.Par.ParDelayFalse := 0;
   A_22_A700Z1.Par.ParTimeoutTrue := 0;
   A_22_A700Z1.Par.ParTimeoutFalse := 0;
   A_22_A700Z1.Par.OutMonTime := 0;
   A_22_A700Z1.Par.OutTransitionTime := 0;
   A_22_A700Z1.Par.OutMonTrue := FALSE;
   A_22_A700Z1.Par.OutMonFalse := FALSE;
   A_22_A700Z1.Par.OutFlagFaultDev := FALSE;
   A_22_A700Z1.Par.OutDelayTime := 0;
   A_22_A800Z1.StCode := 0;
   A_22_A800Z1.InMonTrue := FALSE;
   A_22_A800Z1.InMonFalse := FALSE;
   A_22_A800Z1.InPreAlarmTrue := FALSE;
   A_22_A800Z1.InPreAlarmFalse := FALSE;
   A_22_A800Z1.InStopTrueTime := FALSE;
   A_22_A800Z1.InStopFalseTime := FALSE;
   A_22_A800Z1.InpTrue := FALSE;
   A_22_A800Z1.InpFaultDev := FALSE;
   A_22_A800Z1.CmdRstTrueTime := FALSE;
   A_22_A800Z1.CmdRstFalseTime := FALSE;
   A_22_A800Z1.CmdRunTimeoutTime := FALSE;
   A_22_A800Z1.CmdFaultReset := FALSE;
   A_22_A800Z1.InLocal := FALSE;
   A_22_A800Z1.spare0305 := FALSE;
   A_22_A800Z1.InReport := FALSE;
   A_22_A800Z1.OutTimeoutTime := FALSE;
   A_22_A800Z1.InHWStop := FALSE;
   A_22_A800Z1.InDPFault := FALSE;
   A_22_A800Z1.OutPreAlarmTrue := FALSE;
   A_22_A800Z1.OutPreAlarmFalse := FALSE;
   A_22_A800Z1.OutFlagPos := FALSE;
   A_22_A800Z1.OutFlagNeg := FALSE;
   A_22_A800Z1.OutpFaultReset := FALSE;
   A_22_A800Z1.OutTrue := FALSE;
   A_22_A800Z1.StFalse := FALSE;
   A_22_A800Z1.StCtoTrue := FALSE;
   A_22_A800Z1.StTrue := FALSE;
   A_22_A800Z1.StCtoFalse := FALSE;
   A_22_A800Z1.StFault := FALSE;
   A_22_A800Z1.OutAlarmNrLog := 0;
   A_22_A800Z1.Par.ParObjectNo := 0;
   A_22_A800Z1.Par.ParMsgType := 0;
   A_22_A800Z1.Par.ParHornCode := 0;
   A_22_A800Z1.Par.ParLogOff := FALSE;
   A_22_A800Z1.Par.spare0401 := FALSE;
   A_22_A800Z1.Par.Par2WorkingCond := FALSE;
   A_22_A800Z1.Par.ParFaultRetry := FALSE;
   A_22_A800Z1.Par.ParBinLevel := FALSE;
   A_22_A800Z1.Par.ParDelayChange := 0;
   A_22_A800Z1.Par.ParDelayTrue := 0;
   A_22_A800Z1.Par.ParDelayFalse := 0;
   A_22_A800Z1.Par.ParTimeoutTrue := 0;
   A_22_A800Z1.Par.ParTimeoutFalse := 0;
   A_22_A800Z1.Par.OutMonTime := 0;
   A_22_A800Z1.Par.OutTransitionTime := 0;
   A_22_A800Z1.Par.OutMonTrue := FALSE;
   A_22_A800Z1.Par.OutMonFalse := FALSE;
   A_22_A800Z1.Par.OutFlagFaultDev := FALSE;
   A_22_A800Z1.Par.OutDelayTime := 0;
END_DATA_BLOCK

